LIN {X 0,Y 171.368,Z 489.651,A -85,B 0,C 180,E1 -22896.483,E2 -22896.483} C_VEL
LIN {X 0,Y 171.436,Z 490.117,A -85,B 0,C 180,E1 -22897.2,E2 -22897.2} C_VEL
LIN {X 0,Y 172.205,Z 492.194,A -85,B 0,C 180,E1 -22897.901,E2 -22897.901} C_VEL
LIN {X 0,Y 174.178,Z 494.48,A -85,B 0,C 180,E1 -22898.881,E2 -22898.881} C_VEL
LIN {X 0,Y 175.074,Z 495.303,A -85,B 0,C 180,E1 -22899.298,E2 -22899.298} C_VEL
LIN {X 0,Y 177.261,Z 498.704,A -85,B 0,C 180,E1 -22900.369,E2 -22900.369} C_VEL
LIN {X 0,Y 178.749,Z 500.495,A -85,B 0,C 180,E1 -22901.039,E2 -22901.039} C_VEL
LIN {X 0,Y 181.276,Z 503.935,A -85,B 0,C 180,E1 -22902.154,E2 -22902.154} C_VEL
LIN {X 0,Y 189.16,Z 515.818,A -85,B 0,C 180,E1 -22905.372,E2 -22905.372} C_VEL
LIN {X 0,Y 196.547,Z 528.551,A -85,B 0,C 180,E1 -22908.092,E2 -22908.092} C_VEL
LIN {X 0,Y 202.891,Z 541.51,A -85,B 0,C 180,E1 -22910.279,E2 -22910.279} C_VEL
LIN {X 0,Y 211.2,Z 559.373,A -85,B 0,C 180,E1 -22912.892,E2 -22912.892} C_VEL
LIN {X 0,Y 219.957,Z 574.029,A -85,B 0,C 180,E1 -22915.185,E2 -22915.185} C_VEL
LIN {X 0,Y 227.98,Z 585.278,A -85,B 0,C 180,E1 -22917.037,E2 -22917.037} C_VEL
LIN {X 0,Y 236.394,Z 595.667,A -85,B 0,C 180,E1 -22918.93,E2 -22918.93} C_VEL
LIN {X 0,Y 244.254,Z 604.497,A -85,B 0,C 180,E1 -22920.716,E2 -22920.716} C_VEL
LIN {X 0,Y 253.064,Z 613.517,A -85,B 0,C 180,E1 -22922.703,E2 -22922.703} C_VEL
LIN {X 0,Y 263.679,Z 622.944,A -85,B 0,C 180,E1 -22924.981,E2 -22924.981} C_VEL
LIN {X 0,Y 276.705,Z 633.025,A -85,B 0,C 180,E1 -22927.606,E2 -22927.606} C_VEL
LIN {X 0,Y 290.949,Z 643.204,A -85,B 0,C 180,E1 -22930.392,E2 -22930.392} C_VEL
LIN {X 0,Y 299.892,Z 649.736,A -85,B 0,C 180,E1 -22932.263,E2 -22932.263} C_VEL
LIN {X 0,Y 305.097,Z 653.329,A -85,B 0,C 180,E1 -22933.434,E2 -22933.434} C_VEL
LIN {X 0,Y 312.329,Z 658.424,A -85,B 0,C 180,E1 -22935.36,E2 -22935.36} C_VEL
LIN {X 0,Y 318.766,Z 662.437,A -85,B 0,C 180,E1 -22937.263,E2 -22937.263} C_VEL
LIN {X 0,Y 322.744,Z 665.158,A -85,B 0,C 180,E1 -22938.698,E2 -22938.698} C_VEL
LIN {X 0,Y 327.506,Z 668.458,A -85,B 0,C 180,E1 -22940.777,E2 -22940.777} C_VEL
LIN {X 0,Y 331.235,Z 670.635,A -85,B 0,C 180,E1 -22942.686,E2 -22942.686} C_VEL
LIN {X 0,Y 333.377,Z 671.715,A -85,B 0,C 180,E1 -22943.95,E2 -22943.95} C_VEL
LIN {X 0,Y 335.116,Z 672.498,A -85,B 0,C 180,E1 -22945.188,E2 -22945.188} C_VEL
LIN {X 0,Y 336.568,Z 673.013,A -85,B 0,C 180,E1 -22946.408,E2 -22946.408} C_VEL
LIN {X 0,Y 337.598,Z 673.448,A -85,B 0,C 180,E1 -22947.711,E2 -22947.711} C_VEL
LIN {X 0,Y 338.318,Z 673.7,A -85,B 0,C 180,E1 -22950,E2 -22950} C_VEL
LIN {X 0,Y 338.036,Z 673.676,A -85,B 0,C 180,E1 -22951.191,E2 -22951.191} C_VEL
LIN {X 0,Y 337.502,Z 673.41,A -85,B 0,C 180,E1 -22952.387,E2 -22952.387} C_VEL
LIN {X 0,Y 336.558,Z 672.994,A -85,B 0,C 180,E1 -22953.592,E2 -22953.592} C_VEL
LIN {X 0,Y 335.084,Z 672.488,A -85,B 0,C 180,E1 -22954.812,E2 -22954.812} C_VEL
LIN {X 0,Y 332.493,Z 671.329,A -85,B 0,C 180,E1 -22956.583,E2 -22956.583} C_VEL
LIN {X 0,Y 328.728,Z 669.23,A -85,B 0,C 180,E1 -22958.607,E2 -22958.607} C_VEL
LIN {X 0,Y 324.566,Z 666.489,A -85,B 0,C 180,E1 -22960.529,E2 -22960.529} C_VEL
LIN {X 0,Y 321.225,Z 664.079,A -85,B 0,C 180,E1 -22961.884,E2 -22961.884} C_VEL
LIN {X 0,Y 317.5,Z 661.727,A -85,B 0,C 180,E1 -22963.116,E2 -22963.116} C_VEL
LIN {X 0,Y 312.33,Z 658.43,A -85,B 0,C 180,E1 -22964.64,E2 -22964.64} C_VEL
LIN {X 0,Y 307.138,Z 654.773,A -85,B 0,C 180,E1 -22966.053,E2 -22966.053} C_VEL
LIN {X 0,Y 300.05,Z 649.811,A -85,B 0,C 180,E1 -22967.728,E2 -22967.728} C_VEL
LIN {X 0,Y 289.754,Z 642.358,A -85,B 0,C 180,E1 -22969.85,E2 -22969.85} C_VEL
LIN {X 0,Y 274.478,Z 631.398,A -85,B 0,C 180,E1 -22972.82,E2 -22972.82} C_VEL
LIN {X 0,Y 261.571,Z 621.184,A -85,B 0,C 180,E1 -22975.461,E2 -22975.461} C_VEL
LIN {X 0,Y 249.201,Z 609.815,A -85,B 0,C 180,E1 -22978.147,E2 -22978.147} C_VEL
LIN {X 0,Y 238.841,Z 598.535,A -85,B 0,C 180,E1 -22980.508,E2 -22980.508} C_VEL
LIN {X 0,Y 230.498,Z 588.456,A -85,B 0,C 180,E1 -22982.419,E2 -22982.419} C_VEL
LIN {X 0,Y 222.857,Z 578.314,A -85,B 0,C 180,E1 -22984.131,E2 -22984.131} C_VEL
LIN {X 0,Y 214.033,Z 564.466,A -85,B 0,C 180,E1 -22986.324,E2 -22986.324} C_VEL
LIN {X 0,Y 207.085,Z 551.017,A -85,B 0,C 180,E1 -22988.343,E2 -22988.343} C_VEL
LIN {X 0,Y 200.045,Z 535.481,A -85,B 0,C 180,E1 -22990.686,E2 -22990.686} C_VEL
LIN {X 0,Y 193.982,Z 523.965,A -85,B 0,C 180,E1 -22992.824,E2 -22992.824} C_VEL
LIN {X 0,Y 186.911,Z 512.312,A -85,B 0,C 180,E1 -22995.505,E2 -22995.505} C_VEL
LIN {X 0,Y 180.667,Z 503.29,A -85,B 0,C 180,E1 -22998.099,E2 -22998.099} C_VEL
LIN {X 0,Y 177.863,Z 499.314,A -85,B 0,C 180,E1 -22999.364,E2 -22999.364} C_VEL
LIN {X 0,Y 175.532,Z 496.228,A -85,B 0,C 180,E1 -23000.46,E2 -23000.46} C_VEL
LIN {X 0,Y 174.788,Z 494.891,A -85,B 0,C 180,E1 -23000.844,E2 -23000.844} C_VEL
LIN {X 0,Y 172.504,Z 492.69,A -85,B 0,C 180,E1 -23001.938,E2 -23001.938} C_VEL
LIN {X 0,Y 171.499,Z 490.425,A -85,B 0,C 180,E1 -23002.631,E2 -23002.631} C_VEL
LIN {X 0,Y 171.377,Z 489.669,A -85,B 0,C 180,E1 -23003.336,E2 -23003.336} C_VEL
LIN {X 0,Y 171.381,Z 489.625,A -85,B 0,C 180,E1 -23007.789,E2 -23007.789} C_VEL
LIN {X 0,Y 171.384,Z 489.611,A -85,B 0,C 180,E1 -23010.527,E2 -23010.527} C_VEL
LIN {X 0,Y 171.396,Z 489.63,A -85,B 0,C 180,E1 -23015.797,E2 -23015.797} C_VEL
LIN {X 0,Y 171.502,Z 489.574,A -85,B 0,C 180,E1 -23020.867,E2 -23020.867} C_VEL
LIN {X 0,Y 171.541,Z 489.614,A -85,B 0,C 180,E1 -23025.774,E2 -23025.774} C_VEL
LIN {X 0,Y 171.838,Z 489.529,A -85,B 0,C 180,E1 -23030.588,E2 -23030.588} C_VEL
LIN {X 0,Y 171.774,Z 489.585,A -85,B 0,C 180,E1 -23035.31,E2 -23035.31} C_VEL
LIN {X 0,Y 172.303,Z 489.467,A -85,B 0,C 180,E1 -23040.004,E2 -23040.004} C_VEL
LIN {X 0,Y 171.775,Z 489.588,A -85,B 0,C 180,E1 -23044.697,E2 -23044.697} C_VEL
LIN {X 0,Y 171.84,Z 489.524,A -85,B 0,C 180,E1 -23049.419,E2 -23049.419} C_VEL
LIN {X 0,Y 171.529,Z 489.615,A -85,B 0,C 180,E1 -23054.235,E2 -23054.235} C_VEL
LIN {X 0,Y 171.476,Z 489.578,A -85,B 0,C 180,E1 -23059.498,E2 -23059.498} C_VEL
LIN {X 0,Y 171.404,Z 489.596,A -85,B 0,C 180,E1 -23065.571,E2 -23065.571} C_VEL
LIN {X 0,Y 171.409,Z 489.635,A -85,B 0,C 180,E1 -23070.569,E2 -23070.569} C_VEL
LIN {X 0,Y 171.404,Z 489.723,A -85,B 0,C 180,E1 -23076.301,E2 -23076.301} C_VEL
LIN {X 0,Y 171.544,Z 490.53,A -85,B 0,C 180,E1 -23076.998,E2 -23076.998} C_VEL
LIN {X 0,Y 173.033,Z 493.38,A -85,B 0,C 180,E1 -23077.943,E2 -23077.943} C_VEL
LIN {X 0,Y 175.65,Z 496.732,A -85,B 0,C 180,E1 -23079.23,E2 -23079.23} C_VEL
LIN {X 0,Y 179.466,Z 502.8,A -85,B 0,C 180,E1 -23081.051,E2 -23081.051} C_VEL
LIN {X 0,Y 182.698,Z 508.235,A -85,B 0,C 180,E1 -23082.504,E2 -23082.504} C_VEL
LIN {X 0,Y 189.282,Z 520.227,A -85,B 0,C 180,E1 -23085.251,E2 -23085.251} C_VEL
LIN {X 0,Y 194.403,Z 531.098,A -85,B 0,C 180,E1 -23087.255,E2 -23087.255} C_VEL
LIN {X 0,Y 199.319,Z 543.1,A -85,B 0,C 180,E1 -23089.1,E2 -23089.1} C_VEL
LIN {X 0,Y 200.075,Z 545.841,A -85,B 0,C 180,E1 -23089.413,E2 -23089.413} C_VEL
LIN {X 0,Y 201.512,Z 556.425,A -85,B 0,C 180,E1 -23090.24,E2 -23090.24} C_VEL
LIN {X 0,Y 199.145,Z 597.614,A -85,B 0,C 180,E1 -23091.634,E2 -23091.634} C_VEL
LIN {X 0,Y 197.92,Z 608.393,A -85,B 0,C 180,E1 -23092.223,E2 -23092.223} C_VEL
LIN {X 0,Y 196.28,Z 618.373,A -85,B 0,C 180,E1 -23092.988,E2 -23092.988} C_VEL
LIN {X 0,Y 194.704,Z 626.202,A -85,B 0,C 180,E1 -23093.767,E2 -23093.767} C_VEL
LIN {X 0,Y 192.484,Z 635.344,A -85,B 0,C 180,E1 -23094.896,E2 -23094.896} C_VEL
LIN {X 0,Y 189.963,Z 644.341,A -85,B 0,C 180,E1 -23096.293,E2 -23096.293} C_VEL
LIN {X 0,Y 187.212,Z 653.065,A -85,B 0,C 180,E1 -23097.978,E2 -23097.978} C_VEL
LIN {X 0,Y 184.639,Z 660.483,A -85,B 0,C 180,E1 -23099.713,E2 -23099.713} C_VEL
LIN {X 0,Y 181.263,Z 669.275,A -85,B 0,C 180,E1 -23102.273,E2 -23102.273} C_VEL
LIN {X 0,Y 178.969,Z 675.267,A -85,B 0,C 180,E1 -23104.408,E2 -23104.408} C_VEL
LIN {X 0,Y 176.436,Z 681.58,A -85,B 0,C 180,E1 -23107.147,E2 -23107.147} C_VEL
LIN {X 0,Y 174.148,Z 686.853,A -85,B 0,C 180,E1 -23109.939,E2 -23109.939} C_VEL
LIN {X 0,Y 171.881,Z 691.945,A -85,B 0,C 180,E1 -23113.368,E2 -23113.368} C_VEL
LIN {X 0,Y 170.408,Z 695.916,A -85,B 0,C 180,E1 -23116.889,E2 -23116.889} C_VEL
LIN {X 0,Y 169.423,Z 698.857,A -85,B 0,C 180,E1 -23120.449,E2 -23120.449} C_VEL
LIN {X 0,Y 169.021,Z 700.362,A -85,B 0,C 180,E1 -23122.834,E2 -23122.834} C_VEL
LIN {X 0,Y 168.867,Z 701.898,A -85,B 0,C 180,E1 -23127.615,E2 -23127.615} C_VEL
LIN {X 0,Y 168.971,Z 702.182,A -85,B 0,C 180,E1 -23130,E2 -23130} C_VEL
LIN {X 0,Y 168.87,Z 701.296,A -85,B 0,C 180,E1 -23134.775,E2 -23134.775} C_VEL
LIN {X 0,Y 168.877,Z 701.169,A -85,B 0,C 180,E1 -23135.1,E2 -23135.1} C_VEL
LIN {X 0,Y 168.342,Z 700.396,A -85,B 0,C 180,E1 -23137.08,E2 -23137.08} C_VEL
LIN {X 0,Y 166.004,Z 698.459,A -85,B 0,C 180,E1 -23140.328,E2 -23140.328} C_VEL
LIN {X 0,Y 164.302,Z 696.463,A -85,B 0,C 180,E1 -23142.94,E2 -23142.94} C_VEL
LIN {X 0,Y 163.985,Z 694.593,A -85,B 0,C 180,E1 -23144.901,E2 -23144.901} C_VEL
LIN {X 0,Y 164.176,Z 693.859,A -85,B 0,C 180,E1 -23145.542,E2 -23145.542} C_VEL
LIN {X 0,Y 165.829,Z 690.235,A -85,B 0,C 180,E1 -23148.533,E2 -23148.533} C_VEL
LIN {X 0,Y 168.314,Z 684.658,A -85,B 0,C 180,E1 -23152.073,E2 -23152.073} C_VEL
LIN {X 0,Y 171.157,Z 678.377,A -85,B 0,C 180,E1 -23155.202,E2 -23155.202} C_VEL
LIN {X 0,Y 173.767,Z 672.201,A -85,B 0,C 180,E1 -23157.717,E2 -23157.717} C_VEL
LIN {X 0,Y 177.073,Z 663.985,A -85,B 0,C 180,E1 -23160.4,E2 -23160.4} C_VEL
LIN {X 0,Y 180.029,Z 656.162,A -85,B 0,C 180,E1 -23162.464,E2 -23162.464} C_VEL
LIN {X 0,Y 182.892,Z 648.084,A -85,B 0,C 180,E1 -23164.193,E2 -23164.193} C_VEL
LIN {X 0,Y 185.844,Z 638.326,A -85,B 0,C 180,E1 -23165.884,E2 -23165.884} C_VEL
LIN {X 0,Y 188.077,Z 629.94,A -85,B 0,C 180,E1 -23167.052,E2 -23167.052} C_VEL
LIN {X 0,Y 190.391,Z 619.437,A -85,B 0,C 180,E1 -23168.192,E2 -23168.192} C_VEL
LIN {X 0,Y 192.229,Z 609.145,A -85,B 0,C 180,E1 -23169.011,E2 -23169.011} C_VEL
LIN {X 0,Y 193.567,Z 598.773,A -85,B 0,C 180,E1 -23169.593,E2 -23169.593} C_VEL
LIN {X 0,Y 194.905,Z 576.946,A -85,B 0,C 180,E1 -23170.407,E2 -23170.407} C_VEL
LIN {X 0,Y 195.942,Z 556.279,A -85,B 0,C 180,E1 -23171.126,E2 -23171.126} C_VEL
LIN {X 0,Y 194.549,Z 547.053,A -85,B 0,C 180,E1 -23171.928,E2 -23171.928} C_VEL
LIN {X 0,Y 190.164,Z 535.964,A -85,B 0,C 180,E1 -23173.681,E2 -23173.681} C_VEL
LIN {X 0,Y 185.387,Z 525.465,A -85,B 0,C 180,E1 -23175.663,E2 -23175.663} C_VEL
LIN {X 0,Y 179.255,Z 513.895,A -85,B 0,C 180,E1 -23178.369,E2 -23178.369} C_VEL
LIN {X 0,Y 174.37,Z 505.581,A -85,B 0,C 180,E1 -23180.72,E2 -23180.72} C_VEL
LIN {X 0,Y 171.2,Z 500.576,A -85,B 0,C 180,E1 -23182.36,E2 -23182.36} C_VEL
LIN {X 0,Y 168.626,Z 497.072,A -85,B 0,C 180,E1 -23183.746,E2 -23183.746} C_VEL
LIN {X 0,Y 167.967,Z 495.868,A -85,B 0,C 180,E1 -23184.138,E2 -23184.138} C_VEL
LIN {X 0,Y 165.55,Z 493.655,A -85,B 0,C 180,E1 -23185.468,E2 -23185.468} C_VEL
LIN {X 0,Y 164.421,Z 491.155,A -85,B 0,C 180,E1 -23186.416,E2 -23186.416} C_VEL
LIN {X 0,Y 164.347,Z 490.531,A -85,B 0,C 180,E1 -23187.279,E2 -23187.279} C_VEL
LIN {X 0,Y 164.291,Z 490.484,A -85,B 0,C 180,E1 -23191.926,E2 -23191.926} C_VEL
LIN {X 0,Y 164.358,Z 490.475,A -85,B 0,C 180,E1 -23194.681,E2 -23194.681} C_VEL
LIN {X 0,Y 164.417,Z 490.459,A -85,B 0,C 180,E1 -23200.116,E2 -23200.116} C_VEL
LIN {X 0,Y 164.46,Z 490.486,A -85,B 0,C 180,E1 -23205.14,E2 -23205.14} C_VEL
LIN {X 0,Y 164.759,Z 490.406,A -85,B 0,C 180,E1 -23210.172,E2 -23210.172} C_VEL
LIN {X 0,Y 164.814,Z 490.411,A -85,B 0,C 180,E1 -23212.647,E2 -23212.647} C_VEL
LIN {X 0,Y 165.268,Z 490.343,A -85,B 0,C 180,E1 -23219.996,E2 -23219.996} C_VEL
LIN {X 0,Y 164.813,Z 490.425,A -85,B 0,C 180,E1 -23227.346,E2 -23227.346} C_VEL
LIN {X 0,Y 164.697,Z 490.418,A -85,B 0,C 180,E1 -23231.053,E2 -23231.053} C_VEL
LIN {X 0,Y 164.422,Z 490.466,A -85,B 0,C 180,E1 -23237.406,E2 -23237.406} C_VEL
LIN {X 0,Y 164.414,Z 490.458,A -85,B 0,C 180,E1 -23239.992,E2 -23239.992} C_VEL
LIN {X 0,Y 164.328,Z 490.482,A -85,B 0,C 180,E1 -23246.088,E2 -23246.088} C_VEL
LIN {X 0,Y 164.348,Z 490.498,A -85,B 0,C 180,E1 -23252.362,E2 -23252.362} C_VEL
LIN {X 0,Y 164.353,Z 490.85,A -85,B 0,C 180,E1 -23253.768,E2 -23253.768} C_VEL
LIN {X 0,Y 164.764,Z 492.175,A -85,B 0,C 180,E1 -23254.394,E2 -23254.394} C_VEL
LIN {X 0,Y 166.406,Z 494.696,A -85,B 0,C 180,E1 -23255.421,E2 -23255.421} C_VEL
LIN {X 0,Y 168.271,Z 496.336,A -85,B 0,C 180,E1 -23256.426,E2 -23256.426} C_VEL
LIN {X 0,Y 170.442,Z 499.713,A -85,B 0,C 180,E1 -23257.641,E2 -23257.641} C_VEL
LIN {X 0,Y 172.014,Z 501.392,A -85,B 0,C 180,E1 -23258.43,E2 -23258.43} C_VEL
LIN {X 0,Y 174.717,Z 505.136,A -85,B 0,C 180,E1 -23259.779,E2 -23259.779} C_VEL
LIN {X 0,Y 181.198,Z 514.584,A -85,B 0,C 180,E1 -23262.742,E2 -23262.742} C_VEL
LIN {X 0,Y 187.188,Z 524.201,A -85,B 0,C 180,E1 -23265.216,E2 -23265.216} C_VEL
LIN {X 0,Y 193.294,Z 535.317,A -85,B 0,C 180,E1 -23267.55,E2 -23267.55} C_VEL
LIN {X 0,Y 199.394,Z 548.354,A -85,B 0,C 180,E1 -23269.751,E2 -23269.751} C_VEL
LIN {X 0,Y 206.259,Z 563.313,A -85,B 0,C 180,E1 -23272.01,E2 -23272.01} C_VEL
LIN {X 0,Y 215.082,Z 578.411,A -85,B 0,C 180,E1 -23274.447,E2 -23274.447} C_VEL
LIN {X 0,Y 223.661,Z 590.654,A -85,B 0,C 180,E1 -23276.575,E2 -23276.575} C_VEL
LIN {X 0,Y 233.242,Z 602.662,A -85,B 0,C 180,E1 -23278.992,E2 -23278.992} C_VEL
LIN {X 0,Y 242.719,Z 613.234,A -85,B 0,C 180,E1 -23281.369,E2 -23281.369} C_VEL
LIN {X 0,Y 253.99,Z 624.019,A -85,B 0,C 180,E1 -23284.057,E2 -23284.057} C_VEL
LIN {X 0,Y 267.246,Z 634.657,A -85,B 0,C 180,E1 -23286.981,E2 -23286.981} C_VEL
LIN {X 0,Y 280.808,Z 644.286,A -85,B 0,C 180,E1 -23289.797,E2 -23289.797} C_VEL
LIN {X 0,Y 289.669,Z 650.424,A -85,B 0,C 180,E1 -23291.615,E2 -23291.615} C_VEL
LIN {X 0,Y 298.756,Z 656.783,A -85,B 0,C 180,E1 -23293.603,E2 -23293.603} C_VEL
LIN {X 0,Y 305.451,Z 661.513,A -85,B 0,C 180,E1 -23295.339,E2 -23295.339} C_VEL
LIN {X 0,Y 311.049,Z 665.144,A -85,B 0,C 180,E1 -23296.942,E2 -23296.942} C_VEL
LIN {X 0,Y 315.659,Z 668.041,A -85,B 0,C 180,E1 -23298.441,E2 -23298.441} C_VEL
LIN {X 0,Y 320.614,Z 671.559,A -85,B 0,C 180,E1 -23300.531,E2 -23300.531} C_VEL
LIN {X 0,Y 324.673,Z 674.038,A -85,B 0,C 180,E1 -23302.538,E2 -23302.538} C_VEL
LIN {X 0,Y 326.939,Z 675.216,A -85,B 0,C 180,E1 -23303.83,E2 -23303.83} C_VEL
LIN {X 0,Y 328.818,Z 676.119,A -85,B 0,C 180,E1 -23305.096,E2 -23305.096} C_VEL
LIN {X 0,Y 330.815,Z 676.869,A -85,B 0,C 180,E1 -23306.805,E2 -23306.805} C_VEL
LIN {X 0,Y 331.94,Z 677.388,A -85,B 0,C 180,E1 -23308.787,E2 -23308.787} C_VEL
LIN {X 0,Y 332.268,Z 677.395,A -85,B 0,C 180,E1 -23310,E2 -23310} C_VEL
LIN {X 0,Y 331.956,Z 677.37,A -85,B 0,C 180,E1 -23311.213,E2 -23311.213} C_VEL
LIN {X 0,Y 330.815,Z 676.878,A -85,B 0,C 180,E1 -23313.195,E2 -23313.195} C_VEL
LIN {X 0,Y 328.794,Z 676.11,A -85,B 0,C 180,E1 -23314.905,E2 -23314.905} C_VEL
LIN {X 0,Y 325.649,Z 674.584,A -85,B 0,C 180,E1 -23316.926,E2 -23316.926} C_VEL
LIN {X 0,Y 322.062,Z 672.504,A -85,B 0,C 180,E1 -23318.786,E2 -23318.786} C_VEL
LIN {X 0,Y 319.06,Z 670.533,A -85,B 0,C 180,E1 -23320.149,E2 -23320.149} C_VEL
LIN {X 0,Y 315.62,Z 668.068,A -85,B 0,C 180,E1 -23321.561,E2 -23321.561} C_VEL
LIN {X 0,Y 310.432,Z 664.788,A -85,B 0,C 180,E1 -23323.233,E2 -23323.233} C_VEL
LIN {X 0,Y 305.192,Z 661.373,A -85,B 0,C 180,E1 -23324.73,E2 -23324.73} C_VEL
LIN {X 0,Y 298.775,Z 656.763,A -85,B 0,C 180,E1 -23326.396,E2 -23326.396} C_VEL
LIN {X 0,Y 287.857,Z 649.115,A -85,B 0,C 180,E1 -23328.777,E2 -23328.777} C_VEL
LIN {X 0,Y 274.845,Z 640.119,A -85,B 0,C 180,E1 -23331.433,E2 -23331.433} C_VEL
LIN {X 0,Y 261.888,Z 630.524,A -85,B 0,C 180,E1 -23334.165,E2 -23334.165} C_VEL
LIN {X 0,Y 250.241,Z 620.543,A -85,B 0,C 180,E1 -23336.83,E2 -23336.83} C_VEL
LIN {X 0,Y 241.128,Z 611.5,A -85,B 0,C 180,E1 -23339.034,E2 -23339.034} C_VEL
LIN {X 0,Y 230.967,Z 599.971,A -85,B 0,C 180,E1 -23341.576,E2 -23341.576} C_VEL
LIN {X 0,Y 221.735,Z 588.081,A -85,B 0,C 180,E1 -23343.905,E2 -23343.905} C_VEL
LIN {X 0,Y 211.545,Z 572.787,A -85,B 0,C 180,E1 -23346.479,E2 -23346.479} C_VEL
LIN {X 0,Y 204.033,Z 558.817,A -85,B 0,C 180,E1 -23348.682,E2 -23348.682} C_VEL
LIN {X 0,Y 195.443,Z 539.676,A -85,B 0,C 180,E1 -23351.661,E2 -23351.661} C_VEL
LIN {X 0,Y 189.813,Z 528.782,A -85,B 0,C 180,E1 -23353.761,E2 -23353.761} C_VEL
LIN {X 0,Y 182.873,Z 517.082,A -85,B 0,C 180,E1 -23356.549,E2 -23356.549} C_VEL
LIN {X 0,Y 177.001,Z 508.481,A -85,B 0,C 180,E1 -23359.131,E2 -23359.131} C_VEL
LIN {X 0,Y 174.344,Z 504.736,A -85,B 0,C 180,E1 -23360.395,E2 -23360.395} C_VEL
LIN {X 0,Y 171.31,Z 500.527,A -85,B 0,C 180,E1 -23361.927,E2 -23361.927} C_VEL
LIN {X 0,Y 169.042,Z 497.785,A -85,B 0,C 180,E1 -23363.118,E2 -23363.118} C_VEL
LIN {X 0,Y 167.93,Z 495.858,A -85,B 0,C 180,E1 -23363.767,E2 -23363.767} C_VEL
LIN {X 0,Y 165.685,Z 493.84,A -85,B 0,C 180,E1 -23364.998,E2 -23364.998} C_VEL
LIN {X 0,Y 164.419,Z 491.07,A -85,B 0,C 180,E1 -23366.041,E2 -23366.041} C_VEL
LIN {X 0,Y 164.314,Z 490.518,A -85,B 0,C 180,E1 -23366.929,E2 -23366.929} C_VEL
LIN {X 0,Y 164.349,Z 490.51,A -85,B 0,C 180,E1 -23369.131,E2 -23369.131} C_VEL
LIN {X 0,Y 164.349,Z 490.487,A -85,B 0,C 180,E1 -23374.688,E2 -23374.688} C_VEL
LIN {X 0,Y 164.411,Z 490.458,A -85,B 0,C 180,E1 -23380.121,E2 -23380.121} C_VEL
LIN {X 0,Y 164.469,Z 490.499,A -85,B 0,C 180,E1 -23385.148,E2 -23385.148} C_VEL
LIN {X 0,Y 164.759,Z 490.408,A -85,B 0,C 180,E1 -23390.18,E2 -23390.18} C_VEL
LIN {X 0,Y 164.813,Z 490.425,A -85,B 0,C 180,E1 -23392.654,E2 -23392.654} C_VEL
LIN {X 0,Y 165.268,Z 490.343,A -85,B 0,C 180,E1 -23400.004,E2 -23400.004} C_VEL
LIN {X 0,Y 164.814,Z 490.411,A -85,B 0,C 180,E1 -23407.353,E2 -23407.353} C_VEL
LIN {X 0,Y 164.696,Z 490.423,A -85,B 0,C 180,E1 -23411.051,E2 -23411.051} C_VEL
LIN {X 0,Y 164.417,Z 490.455,A -85,B 0,C 180,E1 -23417.414,E2 -23417.414} C_VEL
LIN {X 0,Y 164.42,Z 490.46,A -85,B 0,C 180,E1 -23420,E2 -23420} C_VEL
LIN {X 0,Y 164.338,Z 490.473,A -85,B 0,C 180,E1 -23426.095,E2 -23426.095} C_VEL
LIN {X 0,Y 164.36,Z 490.509,A -85,B 0,C 180,E1 -23432.369,E2 -23432.369} C_VEL
LIN {X 0,Y 164.371,Z 490.912,A -85,B 0,C 180,E1 -23433.419,E2 -23433.419} C_VEL
LIN {X 0,Y 164.852,Z 492.387,A -85,B 0,C 180,E1 -23434.075,E2 -23434.075} C_VEL
LIN {X 0,Y 166.509,Z 494.761,A -85,B 0,C 180,E1 -23435.087,E2 -23435.087} C_VEL
LIN {X 0,Y 168.197,Z 496.151,A -85,B 0,C 180,E1 -23435.99,E2 -23435.99} C_VEL
LIN {X 0,Y 170.237,Z 499.459,A -85,B 0,C 180,E1 -23437.145,E2 -23437.145} C_VEL
LIN {X 0,Y 172.277,Z 502.221,A -85,B 0,C 180,E1 -23438.207,E2 -23438.207} C_VEL
LIN {X 0,Y 176.131,Z 508.451,A -85,B 0,C 180,E1 -23440.148,E2 -23440.148} C_VEL
LIN {X 0,Y 180.462,Z 516.016,A -85,B 0,C 180,E1 -23442.181,E2 -23442.181} C_VEL
LIN {X 0,Y 186.936,Z 528.657,A -85,B 0,C 180,E1 -23444.987,E2 -23444.987} C_VEL
LIN {X 0,Y 192.82,Z 542.334,A -85,B 0,C 180,E1 -23447.379,E2 -23447.379} C_VEL
LIN {X 0,Y 194.799,Z 548.007,A -85,B 0,C 180,E1 -23448.184,E2 -23448.184} C_VEL
LIN {X 0,Y 196.004,Z 556.741,A -85,B 0,C 180,E1 -23448.912,E2 -23448.912} C_VEL
LIN {X 0,Y 193.657,Z 597.26,A -85,B 0,C 180,E1 -23450.326,E2 -23450.326} C_VEL
LIN {X 0,Y 192.397,Z 608.063,A -85,B 0,C 180,E1 -23450.923,E2 -23450.923} C_VEL
LIN {X 0,Y 190.875,Z 616.913,A -85,B 0,C 180,E1 -23451.587,E2 -23451.587} C_VEL
LIN {X 0,Y 189.006,Z 626.005,A -85,B 0,C 180,E1 -23452.491,E2 -23452.491} C_VEL
LIN {X 0,Y 186.706,Z 635.147,A -85,B 0,C 180,E1 -23453.64,E2 -23453.64} C_VEL
LIN {X 0,Y 184.091,Z 644.145,A -85,B 0,C 180,E1 -23455.065,E2 -23455.065} C_VEL
LIN {X 0,Y 181.225,Z 652.868,A -85,B 0,C 180,E1 -23456.786,E2 -23456.786} C_VEL
LIN {X 0,Y 178.516,Z 660.286,A -85,B 0,C 180,E1 -23458.558,E2 -23458.558} C_VEL
LIN {X 0,Y 174.988,Z 669.078,A -85,B 0,C 180,E1 -23461.187,E2 -23461.187} C_VEL
LIN {X 0,Y 172.568,Z 675.07,A -85,B 0,C 180,E1 -23463.386,E2 -23463.386} C_VEL
LIN {X 0,Y 169.899,Z 681.384,A -85,B 0,C 180,E1 -23466.215,E2 -23466.215} C_VEL
LIN {X 0,Y 167.456,Z 686.656,A -85,B 0,C 180,E1 -23469.1,E2 -23469.1} C_VEL
LIN {X 0,Y 165.073,Z 691.749,A -85,B 0,C 180,E1 -23472.661,E2 -23472.661} C_VEL
LIN {X 0,Y 163.458,Z 695.719,A -85,B 0,C 180,E1 -23476.321,E2 -23476.321} C_VEL
LIN {X 0,Y 162.405,Z 698.66,A -85,B 0,C 180,E1 -23480.032,E2 -23480.032} C_VEL
LIN {X 0,Y 161.962,Z 700.165,A -85,B 0,C 180,E1 -23482.52,E2 -23482.52} C_VEL
LIN {X 0,Y 161.768,Z 701.701,A -85,B 0,C 180,E1 -23487.51,E2 -23487.51} C_VEL
LIN {X 0,Y 161.869,Z 701.985,A -85,B 0,C 180,E1 -23490,E2 -23490} C_VEL
LIN {X 0,Y 161.776,Z 701.099,A -85,B 0,C 180,E1 -23494.984,E2 -23494.984} C_VEL
LIN {X 0,Y 161.98,Z 700.166,A -85,B 0,C 180,E1 -23497.479,E2 -23497.479} C_VEL
LIN {X 0,Y 163.059,Z 696.81,A -85,B 0,C 180,E1 -23502.445,E2 -23502.445} C_VEL
LIN {X 0,Y 164.176,Z 693.859,A -85,B 0,C 180,E1 -23505.542,E2 -23505.542} C_VEL
LIN {X 0,Y 164.476,Z 691.704,A -85,B 0,C 180,E1 -23507.452,E2 -23507.452} C_VEL
LIN {X 0,Y 163.645,Z 687.755,A -85,B 0,C 180,E1 -23510.626,E2 -23510.626} C_VEL
LIN {X 0,Y 163.153,Z 683.225,A -85,B 0,C 180,E1 -23513.713,E2 -23513.713} C_VEL
LIN {X 0,Y 163.948,Z 680,A -85,B 0,C 180,E1 -23515.425,E2 -23515.425} C_VEL
LIN {X 0,Y 167.466,Z 672.003,A -85,B 0,C 180,E1 -23518.856,E2 -23518.856} C_VEL
LIN {X 0,Y 170.965,Z 663.789,A -85,B 0,C 180,E1 -23521.609,E2 -23521.609} C_VEL
LIN {X 0,Y 174.064,Z 655.965,A -85,B 0,C 180,E1 -23523.722,E2 -23523.722} C_VEL
LIN {X 0,Y 177.067,Z 647.888,A -85,B 0,C 180,E1 -23525.484,E2 -23525.484} C_VEL
LIN {X 0,Y 180.143,Z 638.13,A -85,B 0,C 180,E1 -23527.207,E2 -23527.207} C_VEL
LIN {X 0,Y 182.455,Z 629.743,A -85,B 0,C 180,E1 -23528.397,E2 -23528.397} C_VEL
LIN {X 0,Y 184.857,Z 619.241,A -85,B 0,C 180,E1 -23529.554,E2 -23529.554} C_VEL
LIN {X 0,Y 186.808,Z 608.823,A -85,B 0,C 180,E1 -23530.385,E2 -23530.385} C_VEL
LIN {X 0,Y 188.149,Z 598.632,A -85,B 0,C 180,E1 -23530.967,E2 -23530.967} C_VEL
LIN {X 0,Y 189.546,Z 576.839,A -85,B 0,C 180,E1 -23531.796,E2 -23531.796} C_VEL
LIN {X 0,Y 190.585,Z 557.523,A -85,B 0,C 180,E1 -23532.476,E2 -23532.476} C_VEL
LIN {X 0,Y 189.405,Z 549.639,A -85,B 0,C 180,E1 -23533.2,E2 -23533.2} C_VEL
LIN {X 0,Y 184.565,Z 537.416,A -85,B 0,C 180,E1 -23535.274,E2 -23535.274} C_VEL
LIN {X 0,Y 180.217,Z 527.991,A -85,B 0,C 180,E1 -23537.215,E2 -23537.215} C_VEL
LIN {X 0,Y 173.933,Z 515.984,A -85,B 0,C 180,E1 -23540.235,E2 -23540.235} C_VEL
LIN {X 0,Y 170.407,Z 510.142,A -85,B 0,C 180,E1 -23542.061,E2 -23542.061} C_VEL
LIN {X 0,Y 167.874,Z 506.005,A -85,B 0,C 180,E1 -23543.465,E2 -23543.465} C_VEL
LIN {X 0,Y 164.74,Z 501.67,A -85,B 0,C 180,E1 -23545.274,E2 -23545.274} C_VEL
LIN {X 0,Y 162.18,Z 498.652,A -85,B 0,C 180,E1 -23546.828,E2 -23546.828} C_VEL
LIN {X 0,Y 161.169,Z 496.857,A -85,B 0,C 180,E1 -23547.523,E2 -23547.523} C_VEL
LIN {X 0,Y 158.82,Z 494.949,A -85,B 0,C 180,E1 -23549.032,E2 -23549.032} C_VEL
LIN {X 0,Y 157.364,Z 492.026,A -85,B 0,C 180,E1 -23550.388,E2 -23550.388} C_VEL
LIN {X 0,Y 157.237,Z 491.432,A -85,B 0,C 180,E1 -23551.279,E2 -23551.279} C_VEL
LIN {X 0,Y 157.267,Z 491.377,A -85,B 0,C 180,E1 -23556.281,E2 -23556.281} C_VEL
LIN {X 0,Y 157.36,Z 491.341,A -85,B 0,C 180,E1 -23559.7,E2 -23559.7} C_VEL
LIN {X 0,Y 157.396,Z 491.35,A -85,B 0,C 180,E1 -23564.456,E2 -23564.456} C_VEL
LIN {X 0,Y 157.681,Z 491.289,A -85,B 0,C 180,E1 -23569.726,E2 -23569.726} C_VEL
LIN {X 0,Y 157.753,Z 491.285,A -85,B 0,C 180,E1 -23572.315,E2 -23572.315} C_VEL
LIN {X 0,Y 158.23,Z 491.218,A -85,B 0,C 180,E1 -23579.996,E2 -23579.996} C_VEL
LIN {X 0,Y 157.752,Z 491.298,A -85,B 0,C 180,E1 -23587.677,E2 -23587.677} C_VEL
LIN {X 0,Y 157.626,Z 491.299,A -85,B 0,C 180,E1 -23591.219,E2 -23591.219} C_VEL
LIN {X 0,Y 157.402,Z 491.371,A -85,B 0,C 180,E1 -23595.535,E2 -23595.535} C_VEL
LIN {X 0,Y 157.297,Z 491.351,A -85,B 0,C 180,E1 -23600.938,E2 -23600.938} C_VEL
LIN {X 0,Y 157.259,Z 491.358,A -85,B 0,C 180,E1 -23606.645,E2 -23606.645} C_VEL
LIN {X 0,Y 157.278,Z 491.657,A -85,B 0,C 180,E1 -23609.621,E2 -23609.621} C_VEL
LIN {X 0,Y 157.592,Z 492.786,A -85,B 0,C 180,E1 -23610.385,E2 -23610.385} C_VEL
LIN {X 0,Y 159.197,Z 495.38,A -85,B 0,C 180,E1 -23611.617,E2 -23611.617} C_VEL
LIN {X 0,Y 161.459,Z 497.163,A -85,B 0,C 180,E1 -23613.051,E2 -23613.051} C_VEL
LIN {X 0,Y 163.482,Z 500.487,A -85,B 0,C 180,E1 -23614.388,E2 -23614.388} C_VEL
LIN {X 0,Y 165.501,Z 502.633,A -85,B 0,C 180,E1 -23615.561,E2 -23615.561} C_VEL
LIN {X 0,Y 168.085,Z 506.198,A -85,B 0,C 180,E1 -23617.034,E2 -23617.034} C_VEL
LIN {X 0,Y 172.906,Z 512.986,A -85,B 0,C 180,E1 -23619.554,E2 -23619.554} C_VEL
LIN {X 0,Y 177.99,Z 520.544,A -85,B 0,C 180,E1 -23621.959,E2 -23621.959} C_VEL
LIN {X 0,Y 183.619,Z 529.846,A -85,B 0,C 180,E1 -23624.404,E2 -23624.404} C_VEL
LIN {X 0,Y 189.395,Z 540.762,A -85,B 0,C 180,E1 -23626.733,E2 -23626.733} C_VEL
LIN {X 0,Y 194.728,Z 552.601,A -85,B 0,C 180,E1 -23628.775,E2 -23628.775} C_VEL
LIN {X 0,Y 201.859,Z 568.247,A -85,B 0,C 180,E1 -23631.242,E2 -23631.242} C_VEL
LIN {X 0,Y 210.51,Z 583.179,A -85,B 0,C 180,E1 -23633.746,E2 -23633.746} C_VEL
LIN {X 0,Y 218.276,Z 594.692,A -85,B 0,C 180,E1 -23635.897,E2 -23635.897} C_VEL
LIN {X 0,Y 226.162,Z 605.048,A -85,B 0,C 180,E1 -23638.111,E2 -23638.111} C_VEL
LIN {X 0,Y 234.418,Z 614.641,A -85,B 0,C 180,E1 -23640.387,E2 -23640.387} C_VEL
LIN {X 0,Y 242.814,Z 623.364,A -85,B 0,C 180,E1 -23642.63,E2 -23642.63} C_VEL
LIN {X 0,Y 254.728,Z 633.732,A -85,B 0,C 180,E1 -23645.564,E2 -23645.564} C_VEL
LIN {X 0,Y 269.029,Z 644.182,A -85,B 0,C 180,E1 -23648.781,E2 -23648.781} C_VEL
LIN {X 0,Y 281.628,Z 652.561,A -85,B 0,C 180,E1 -23651.484,E2 -23651.484} C_VEL
LIN {X 0,Y 292.553,Z 660.061,A -85,B 0,C 180,E1 -23653.919,E2 -23653.919} C_VEL
LIN {X 0,Y 299.534,Z 664.986,A -85,B 0,C 180,E1 -23655.704,E2 -23655.704} C_VEL
LIN {X 0,Y 304.733,Z 668.357,A -85,B 0,C 180,E1 -23657.162,E2 -23657.162} C_VEL
LIN {X 0,Y 309.727,Z 671.52,A -85,B 0,C 180,E1 -23658.772,E2 -23658.772} C_VEL
LIN {X 0,Y 313.619,Z 674.292,A -85,B 0,C 180,E1 -23660.389,E2 -23660.389} C_VEL
LIN {X 0,Y 318.723,Z 677.455,A -85,B 0,C 180,E1 -23662.851,E2 -23662.851} C_VEL
LIN {X 0,Y 322.189,Z 679.196,A -85,B 0,C 180,E1 -23664.994,E2 -23664.994} C_VEL
LIN {X 0,Y 323.932,Z 679.922,A -85,B 0,C 180,E1 -23666.344,E2 -23666.344} C_VEL
LIN {X 0,Y 325.013,Z 680.344,A -85,B 0,C 180,E1 -23667.521,E2 -23667.521} C_VEL
LIN {X 0,Y 325.623,Z 680.637,A -85,B 0,C 180,E1 -23668.763,E2 -23668.763} C_VEL
LIN {X 0,Y 325.956,Z 680.664,A -85,B 0,C 180,E1 -23670,E2 -23670} C_VEL
LIN {X 0,Y 325.634,Z 680.624,A -85,B 0,C 180,E1 -23671.237,E2 -23671.237} C_VEL
LIN {X 0,Y 325.013,Z 680.333,A -85,B 0,C 180,E1 -23672.479,E2 -23672.479} C_VEL
LIN {X 0,Y 323.839,Z 679.87,A -85,B 0,C 180,E1 -23673.733,E2 -23673.733} C_VEL
LIN {X 0,Y 322.172,Z 679.197,A -85,B 0,C 180,E1 -23675.006,E2 -23675.006} C_VEL
LIN {X 0,Y 318.703,Z 677.482,A -85,B 0,C 180,E1 -23677.121,E2 -23677.121} C_VEL
LIN {X 0,Y 314.988,Z 675.237,A -85,B 0,C 180,E1 -23678.985,E2 -23678.985} C_VEL
LIN {X 0,Y 311.78,Z 673.038,A -85,B 0,C 180,E1 -23680.389,E2 -23680.389} C_VEL
LIN {X 0,Y 307.878,Z 670.331,A -85,B 0,C 180,E1 -23681.855,E2 -23681.855} C_VEL
LIN {X 0,Y 302.651,Z 667.041,A -85,B 0,C 180,E1 -23683.427,E2 -23683.427} C_VEL
LIN {X 0,Y 296.488,Z 662.798,A -85,B 0,C 180,E1 -23685.114,E2 -23685.114} C_VEL
LIN {X 0,Y 289.821,Z 658.167,A -85,B 0,C 180,E1 -23686.706,E2 -23686.706} C_VEL
LIN {X 0,Y 278.836,Z 650.743,A -85,B 0,C 180,E1 -23689.127,E2 -23689.127} C_VEL
LIN {X 0,Y 263.564,Z 640.349,A -85,B 0,C 180,E1 -23692.419,E2 -23692.419} C_VEL
LIN {X 0,Y 252.116,Z 631.599,A -85,B 0,C 180,E1 -23695.051,E2 -23695.051} C_VEL
LIN {X 0,Y 241.185,Z 621.822,A -85,B 0,C 180,E1 -23697.79,E2 -23697.79} C_VEL
LIN {X 0,Y 230.712,Z 610.495,A -85,B 0,C 180,E1 -23700.621,E2 -23700.621} C_VEL
LIN {X 0,Y 221.954,Z 599.646,A -85,B 0,C 180,E1 -23703.065,E2 -23703.065} C_VEL
LIN {X 0,Y 214.414,Z 589.166,A -85,B 0,C 180,E1 -23705.181,E2 -23705.181} C_VEL
LIN {X 0,Y 205.872,Z 575.535,A -85,B 0,C 180,E1 -23707.545,E2 -23707.545} C_VEL
LIN {X 0,Y 198.966,Z 562.296,A -85,B 0,C 180,E1 -23709.708,E2 -23709.708} C_VEL
LIN {X 0,Y 190.822,Z 543.776,A -85,B 0,C 180,E1 -23712.71,E2 -23712.71} C_VEL
LIN {X 0,Y 185.41,Z 533.084,A -85,B 0,C 180,E1 -23714.856,E2 -23714.856} C_VEL
LIN {X 0,Y 179.132,Z 522.27,A -85,B 0,C 180,E1 -23717.533,E2 -23717.533} C_VEL
LIN {X 0,Y 173.232,Z 513.452,A -85,B 0,C 180,E1 -23720.285,E2 -23720.285} C_VEL
LIN {X 0,Y 170.673,Z 509.812,A -85,B 0,C 180,E1 -23721.58,E2 -23721.58} C_VEL
LIN {X 0,Y 167.965,Z 506.081,A -85,B 0,C 180,E1 -23723.029,E2 -23723.029} C_VEL
LIN {X 0,Y 165.409,Z 502.425,A -85,B 0,C 180,E1 -23724.498,E2 -23724.498} C_VEL
LIN {X 0,Y 162.256,Z 498.764,A -85,B 0,C 180,E1 -23726.39,E2 -23726.39} C_VEL
LIN {X 0,Y 161.135,Z 496.856,A -85,B 0,C 180,E1 -23727.153,E2 -23727.153} C_VEL
LIN {X 0,Y 158.693,Z 494.791,A -85,B 0,C 180,E1 -23728.732,E2 -23728.732} C_VEL
LIN {X 0,Y 157.355,Z 491.978,A -85,B 0,C 180,E1 -23730.027,E2 -23730.027} C_VEL
LIN {X 0,Y 157.227,Z 491.408,A -85,B 0,C 180,E1 -23731.286,E2 -23731.286} C_VEL
LIN {X 0,Y 157.259,Z 491.397,A -85,B 0,C 180,E1 -23736.288,E2 -23736.288} C_VEL
LIN {X 0,Y 157.353,Z 491.338,A -85,B 0,C 180,E1 -23739.707,E2 -23739.707} C_VEL
LIN {X 0,Y 157.402,Z 491.371,A -85,B 0,C 180,E1 -23744.465,E2 -23744.465} C_VEL
LIN {X 0,Y 157.682,Z 491.288,A -85,B 0,C 180,E1 -23749.734,E2 -23749.734} C_VEL
LIN {X 0,Y 157.752,Z 491.298,A -85,B 0,C 180,E1 -23752.323,E2 -23752.323} C_VEL
LIN {X 0,Y 158.23,Z 491.218,A -85,B 0,C 180,E1 -23760.004,E2 -23760.004} C_VEL
LIN {X 0,Y 157.753,Z 491.285,A -85,B 0,C 180,E1 -23767.685,E2 -23767.685} C_VEL
LIN {X 0,Y 157.626,Z 491.304,A -85,B 0,C 180,E1 -23771.219,E2 -23771.219} C_VEL
LIN {X 0,Y 157.396,Z 491.35,A -85,B 0,C 180,E1 -23775.544,E2 -23775.544} C_VEL
LIN {X 0,Y 157.303,Z 491.357,A -85,B 0,C 180,E1 -23780.946,E2 -23780.946} C_VEL
LIN {X 0,Y 157.269,Z 491.352,A -85,B 0,C 180,E1 -23786.652,E2 -23786.652} C_VEL
LIN {X 0,Y 157.283,Z 491.658,A -85,B 0,C 180,E1 -23789.261,E2 -23789.261} C_VEL
LIN {X 0,Y 157.615,Z 492.844,A -85,B 0,C 180,E1 -23790.02,E2 -23790.02} C_VEL
LIN {X 0,Y 159.232,Z 495.422,A -85,B 0,C 180,E1 -23791.253,E2 -23791.253} C_VEL
LIN {X 0,Y 161.583,Z 497.458,A -85,B 0,C 180,E1 -23792.753,E2 -23792.753} C_VEL
LIN {X 0,Y 163.589,Z 500.569,A -85,B 0,C 180,E1 -23794.06,E2 -23794.06} C_VEL
LIN {X 0,Y 165.378,Z 502.391,A -85,B 0,C 180,E1 -23795.095,E2 -23795.095} C_VEL
LIN {X 0,Y 168.077,Z 506.278,A -85,B 0,C 180,E1 -23796.647,E2 -23796.647} C_VEL
LIN {X 0,Y 172.43,Z 513.44,A -85,B 0,C 180,E1 -23799.001,E2 -23799.001} C_VEL
LIN {X 0,Y 176.489,Z 520.707,A -85,B 0,C 180,E1 -23801.032,E2 -23801.032} C_VEL
LIN {X 0,Y 182.602,Z 532.892,A -85,B 0,C 180,E1 -23803.855,E2 -23803.855} C_VEL
LIN {X 0,Y 188.2,Z 546.423,A -85,B 0,C 180,E1 -23806.291,E2 -23806.291} C_VEL
LIN {X 0,Y 189.722,Z 550.794,A -85,B 0,C 180,E1 -23806.947,E2 -23806.947} C_VEL
LIN {X 0,Y 190.632,Z 558.719,A -85,B 0,C 180,E1 -23807.597,E2 -23807.597} C_VEL
LIN {X 0,Y 188.251,Z 597.07,A -85,B 0,C 180,E1 -23808.947,E2 -23808.947} C_VEL
LIN {X 0,Y 186.956,Z 607.807,A -85,B 0,C 180,E1 -23809.55,E2 -23809.55} C_VEL
LIN {X 0,Y 185.374,Z 616.718,A -85,B 0,C 180,E1 -23810.225,E2 -23810.225} C_VEL
LIN {X 0,Y 183.42,Z 625.809,A -85,B 0,C 180,E1 -23811.14,E2 -23811.14} C_VEL
LIN {X 0,Y 181.042,Z 634.951,A -85,B 0,C 180,E1 -23812.309,E2 -23812.309} C_VEL
LIN {X 0,Y 178.308,Z 643.948,A -85,B 0,C 180,E1 -23813.757,E2 -23813.757} C_VEL
LIN {X 0,Y 175.315,Z 652.672,A -85,B 0,C 180,E1 -23815.512,E2 -23815.512} C_VEL
LIN {X 0,Y 172.469,Z 660.089,A -85,B 0,C 180,E1 -23817.322,E2 -23817.322} C_VEL
LIN {X 0,Y 168.775,Z 668.881,A -85,B 0,C 180,E1 -23820.021,E2 -23820.021} C_VEL
LIN {X 0,Y 166.221,Z 674.873,A -85,B 0,C 180,E1 -23822.284,E2 -23822.284} C_VEL
LIN {X 0,Y 163.388,Z 681.186,A -85,B 0,C 180,E1 -23825.204,E2 -23825.204} C_VEL
LIN {X 0,Y 160.794,Z 686.458,A -85,B 0,C 180,E1 -23828.191,E2 -23828.191} C_VEL
LIN {X 0,Y 158.298,Z 691.552,A -85,B 0,C 180,E1 -23831.894,E2 -23831.894} C_VEL
LIN {X 0,Y 156.532,Z 695.522,A -85,B 0,C 180,E1 -23835.704,E2 -23835.704} C_VEL
LIN {X 0,Y 155.407,Z 698.464,A -85,B 0,C 180,E1 -23839.578,E2 -23839.578} C_VEL
LIN {X 0,Y 154.923,Z 699.969,A -85,B 0,C 180,E1 -23842.178,E2 -23842.178} C_VEL
LIN {X 0,Y 154.673,Z 701.505,A -85,B 0,C 180,E1 -23847.396,E2 -23847.396} C_VEL
LIN {X 0,Y 154.782,Z 701.789,A -85,B 0,C 180,E1 -23850,E2 -23850} C_VEL
LIN {X 0,Y 154.703,Z 700.903,A -85,B 0,C 180,E1 -23855.213,E2 -23855.213} C_VEL
LIN {X 0,Y 154.937,Z 699.969,A -85,B 0,C 180,E1 -23857.821,E2 -23857.821} C_VEL
LIN {X 0,Y 156.088,Z 696.613,A -85,B 0,C 180,E1 -23863.01,E2 -23863.01} C_VEL
LIN {X 0,Y 157.615,Z 692.981,A -85,B 0,C 180,E1 -23866.848,E2 -23866.848} C_VEL
LIN {X 0,Y 159.934,Z 688.249,A -85,B 0,C 180,E1 -23870.582,E2 -23870.582} C_VEL
LIN {X 0,Y 162.849,Z 682.279,A -85,B 0,C 180,E1 -23874.204,E2 -23874.204} C_VEL
LIN {X 0,Y 163.948,Z 680,A -85,B 0,C 180,E1 -23875.425,E2 -23875.425} C_VEL
LIN {X 0,Y 164.807,Z 676.605,A -85,B 0,C 180,E1 -23877.067,E2 -23877.067} C_VEL
LIN {X 0,Y 164.848,Z 670.82,A -85,B 0,C 180,E1 -23879.847,E2 -23879.847} C_VEL
LIN {X 0,Y 165.145,Z 664.579,A -85,B 0,C 180,E1 -23882.499,E2 -23882.499} C_VEL
LIN {X 0,Y 166.371,Z 660.272,A -85,B 0,C 180,E1 -23883.886,E2 -23883.886} C_VEL
LIN {X 0,Y 170.868,Z 649.003,A -85,B 0,C 180,E1 -23886.612,E2 -23886.612} C_VEL
LIN {X 0,Y 174.072,Z 639.523,A -85,B 0,C 180,E1 -23888.37,E2 -23888.37} C_VEL
LIN {X 0,Y 176.939,Z 629.547,A -85,B 0,C 180,E1 -23889.827,E2 -23889.827} C_VEL
LIN {X 0,Y 179.431,Z 619.044,A -85,B 0,C 180,E1 -23891,E2 -23891} C_VEL
LIN {X 0,Y 181.393,Z 609.039,A -85,B 0,C 180,E1 -23891.811,E2 -23891.811} C_VEL
LIN {X 0,Y 182.858,Z 597.896,A -85,B 0,C 180,E1 -23892.461,E2 -23892.461} C_VEL
LIN {X 0,Y 184.528,Z 573.459,A -85,B 0,C 180,E1 -23893.371,E2 -23893.371} C_VEL
LIN {X 0,Y 185.351,Z 558.629,A -85,B 0,C 180,E1 -23893.906,E2 -23893.906} C_VEL
LIN {X 0,Y 184.399,Z 552.465,A -85,B 0,C 180,E1 -23894.518,E2 -23894.518} C_VEL
LIN {X 0,Y 179.211,Z 539.178,A -85,B 0,C 180,E1 -23896.916,E2 -23896.916} C_VEL
LIN {X 0,Y 174.112,Z 528.451,A -85,B 0,C 180,E1 -23899.388,E2 -23899.388} C_VEL
LIN {X 0,Y 169.562,Z 519.798,A -85,B 0,C 180,E1 -23901.776,E2 -23901.776} C_VEL
LIN {X 0,Y 165.111,Z 512.074,A -85,B 0,C 180,E1 -23904.326,E2 -23904.326} C_VEL
LIN {X 0,Y 161.762,Z 507.476,A -85,B 0,C 180,E1 -23906.358,E2 -23906.358} C_VEL
LIN {X 0,Y 159.134,Z 504,A -85,B 0,C 180,E1 -23908.085,E2 -23908.085} C_VEL
LIN {X 0,Y 158.275,Z 502.9,A -85,B 0,C 180,E1 -23908.677,E2 -23908.677} C_VEL
LIN {X 0,Y 155.8,Z 500.269,A -85,B 0,C 180,E1 -23910.433,E2 -23910.433} C_VEL
LIN {X 0,Y 154.545,Z 497.966,A -85,B 0,C 180,E1 -23911.474,E2 -23911.474} C_VEL
LIN {X 0,Y 151.987,Z 496.1,A -85,B 0,C 180,E1 -23913.478,E2 -23913.478} C_VEL
LIN {X 0,Y 150.538,Z 493.71,A -85,B 0,C 180,E1 -23914.893,E2 -23914.893} C_VEL
LIN {X 0,Y 150.239,Z 492.531,A -85,B 0,C 180,E1 -23915.834,E2 -23915.834} C_VEL
LIN {X 0,Y 150.296,Z 492.211,A -85,B 0,C 180,E1 -23920.889,E2 -23920.889} C_VEL
LIN {X 0,Y 150.395,Z 492.243,A -85,B 0,C 180,E1 -23926.484,E2 -23926.484} C_VEL
LIN {X 0,Y 150.601,Z 492.173,A -85,B 0,C 180,E1 -23929.238,E2 -23929.238} C_VEL
LIN {X 0,Y 150.676,Z 492.163,A -85,B 0,C 180,E1 -23931.952,E2 -23931.952} C_VEL
LIN {X 0,Y 151.191,Z 492.094,A -85,B 0,C 180,E1 -23939.996,E2 -23939.996} C_VEL
LIN {X 0,Y 150.675,Z 492.173,A -85,B 0,C 180,E1 -23948.04,E2 -23948.04} C_VEL
LIN {X 0,Y 150.569,Z 492.178,A -85,B 0,C 180,E1 -23951.423,E2 -23951.423} C_VEL
LIN {X 0,Y 150.306,Z 492.238,A -85,B 0,C 180,E1 -23956.288,E2 -23956.288} C_VEL
LIN {X 0,Y 150.276,Z 492.222,A -85,B 0,C 180,E1 -23960.718,E2 -23960.718} C_VEL
LIN {X 0,Y 150.221,Z 492.544,A -85,B 0,C 180,E1 -23964.62,E2 -23964.62} C_VEL
LIN {X 0,Y 150.53,Z 493.696,A -85,B 0,C 180,E1 -23965.488,E2 -23965.488} C_VEL
LIN {X 0,Y 152.154,Z 496.309,A -85,B 0,C 180,E1 -23967.057,E2 -23967.057} C_VEL
LIN {X 0,Y 154.791,Z 498.354,A -85,B 0,C 180,E1 -23969.117,E2 -23969.117} C_VEL
LIN {X 0,Y 156.742,Z 501.539,A -85,B 0,C 180,E1 -23970.666,E2 -23970.666} C_VEL
LIN {X 0,Y 158.906,Z 503.572,A -85,B 0,C 180,E1 -23972.137,E2 -23972.137} C_VEL
LIN {X 0,Y 161.51,Z 507.252,A -85,B 0,C 180,E1 -23973.88,E2 -23973.88} C_VEL
LIN {X 0,Y 162.978,Z 509.115,A -85,B 0,C 180,E1 -23974.788,E2 -23974.788} C_VEL
LIN {X 0,Y 166.411,Z 513.885,A -85,B 0,C 180,E1 -23976.806,E2 -23976.806} C_VEL
LIN {X 0,Y 171.509,Z 521.273,A -85,B 0,C 180,E1 -23979.521,E2 -23979.521} C_VEL
LIN {X 0,Y 177.993,Z 531.767,A -85,B 0,C 180,E1 -23982.622,E2 -23982.622} C_VEL
LIN {X 0,Y 184.072,Z 543.159,A -85,B 0,C 180,E1 -23985.272,E2 -23985.272} C_VEL
LIN {X 0,Y 189.756,Z 555.786,A -85,B 0,C 180,E1 -23987.598,E2 -23987.598} C_VEL
LIN {X 0,Y 196.355,Z 570.897,A -85,B 0,C 180,E1 -23990.056,E2 -23990.056} C_VEL
LIN {X 0,Y 204.632,Z 585.908,A -85,B 0,C 180,E1 -23992.677,E2 -23992.677} C_VEL
LIN {X 0,Y 211.511,Z 596.726,A -85,B 0,C 180,E1 -23994.798,E2 -23994.798} C_VEL
LIN {X 0,Y 218.17,Z 606.024,A -85,B 0,C 180,E1 -23996.876,E2 -23996.876} C_VEL
LIN {X 0,Y 226.054,Z 615.945,A -85,B 0,C 180,E1 -23999.313,E2 -23999.313} C_VEL
LIN {X 0,Y 234.945,Z 625.613,A -85,B 0,C 180,E1 -24001.932,E2 -24001.932} C_VEL
LIN {X 0,Y 246.23,Z 635.81,A -85,B 0,C 180,E1 -24004.98,E2 -24004.98} C_VEL
LIN {X 0,Y 257.971,Z 644.659,A -85,B 0,C 180,E1 -24007.853,E2 -24007.853} C_VEL
LIN {X 0,Y 268.721,Z 651.822,A -85,B 0,C 180,E1 -24010.301,E2 -24010.301} C_VEL
LIN {X 0,Y 279.627,Z 658.8,A -85,B 0,C 180,E1 -24012.75,E2 -24012.75} C_VEL
LIN {X 0,Y 287.841,Z 664.098,A -85,B 0,C 180,E1 -24014.661,E2 -24014.661} C_VEL
LIN {X 0,Y 293.557,Z 668.036,A -85,B 0,C 180,E1 -24016.149,E2 -24016.149} C_VEL
LIN {X 0,Y 299.461,Z 671.891,A -85,B 0,C 180,E1 -24017.806,E2 -24017.806} C_VEL
LIN {X 0,Y 304.101,Z 674.865,A -85,B 0,C 180,E1 -24019.346,E2 -24019.346} C_VEL
LIN {X 0,Y 307.578,Z 677.316,A -85,B 0,C 180,E1 -24020.796,E2 -24020.796} C_VEL
LIN {X 0,Y 311.699,Z 679.876,A -85,B 0,C 180,E1 -24022.765,E2 -24022.765} C_VEL
LIN {X 0,Y 315.277,Z 681.806,A -85,B 0,C 180,E1 -24024.884,E2 -24024.884} C_VEL
LIN {X 0,Y 317.041,Z 682.548,A -85,B 0,C 180,E1 -24026.187,E2 -24026.187} C_VEL
LIN {X 0,Y 318.356,Z 683.048,A -85,B 0,C 180,E1 -24027.469,E2 -24027.469} C_VEL
LIN {X 0,Y 319.06,Z 683.372,A -85,B 0,C 180,E1 -24028.738,E2 -24028.738} C_VEL
LIN {X 0,Y 319.431,Z 683.427,A -85,B 0,C 180,E1 -24030,E2 -24030} C_VEL
LIN {X 0,Y 319.068,Z 683.365,A -85,B 0,C 180,E1 -24031.262,E2 -24031.262} C_VEL
LIN {X 0,Y 318.356,Z 683.046,A -85,B 0,C 180,E1 -24032.531,E2 -24032.531} C_VEL
LIN {X 0,Y 316.971,Z 682.519,A -85,B 0,C 180,E1 -24033.878,E2 -24033.878} C_VEL
LIN {X 0,Y 315.264,Z 681.812,A -85,B 0,C 180,E1 -24035.116,E2 -24035.116} C_VEL
LIN {X 0,Y 311.676,Z 679.929,A -85,B 0,C 180,E1 -24037.201,E2 -24037.201} C_VEL
LIN {X 0,Y 307.556,Z 677.303,A -85,B 0,C 180,E1 -24039.204,E2 -24039.204} C_VEL
LIN {X 0,Y 304.069,Z 674.859,A -85,B 0,C 180,E1 -24040.655,E2 -24040.655} C_VEL
LIN {X 0,Y 299.399,Z 671.87,A -85,B 0,C 180,E1 -24042.196,E2 -24042.196} C_VEL
LIN {X 0,Y 292.278,Z 667.133,A -85,B 0,C 180,E1 -24044.215,E2 -24044.215} C_VEL
LIN {X 0,Y 285.114,Z 662.279,A -85,B 0,C 180,E1 -24045.994,E2 -24045.994} C_VEL
LIN {X 0,Y 274.173,Z 655.237,A -85,B 0,C 180,E1 -24048.489,E2 -24048.489} C_VEL
LIN {X 0,Y 263.325,Z 648.262,A -85,B 0,C 180,E1 -24050.92,E2 -24050.92} C_VEL
LIN {X 0,Y 251.012,Z 639.577,A -85,B 0,C 180,E1 -24053.814,E2 -24053.814} C_VEL
LIN {X 0,Y 240.819,Z 631.1,A -85,B 0,C 180,E1 -24056.45,E2 -24056.45} C_VEL
LIN {X 0,Y 231.69,Z 622.123,A -85,B 0,C 180,E1 -24059.034,E2 -24059.034} C_VEL
LIN {X 0,Y 221.723,Z 610.617,A -85,B 0,C 180,E1 -24062.023,E2 -24062.023} C_VEL
LIN {X 0,Y 213.6,Z 599.738,A -85,B 0,C 180,E1 -24064.55,E2 -24064.55} C_VEL
LIN {X 0,Y 207.535,Z 590.449,A -85,B 0,C 180,E1 -24066.466,E2 -24066.466} C_VEL
LIN {X 0,Y 200.665,Z 579.043,A -85,B 0,C 180,E1 -24068.547,E2 -24068.547} C_VEL
LIN {X 0,Y 193.42,Z 564.629,A -85,B 0,C 180,E1 -24070.983,E2 -24070.983} C_VEL
LIN {X 0,Y 186.355,Z 547.997,A -85,B 0,C 180,E1 -24073.778,E2 -24073.778} C_VEL
LIN {X 0,Y 181.096,Z 537.426,A -85,B 0,C 180,E1 -24075.996,E2 -24075.996} C_VEL
LIN {X 0,Y 175.144,Z 526.984,A -85,B 0,C 180,E1 -24078.699,E2 -24078.699} C_VEL
LIN {X 0,Y 169.933,Z 518.99,A -85,B 0,C 180,E1 -24081.284,E2 -24081.284} C_VEL
LIN {X 0,Y 165.253,Z 512.147,A -85,B 0,C 180,E1 -24083.864,E2 -24083.864} C_VEL
LIN {X 0,Y 162.546,Z 508.374,A -85,B 0,C 180,E1 -24085.49,E2 -24085.49} C_VEL
LIN {X 0,Y 159.39,Z 504.453,A -85,B 0,C 180,E1 -24087.512,E2 -24087.512} C_VEL
LIN {X 0,Y 158.4,Z 503.002,A -85,B 0,C 180,E1 -24088.206,E2 -24088.206} C_VEL
LIN {X 0,Y 155.939,Z 500.486,A -85,B 0,C 180,E1 -24089.935,E2 -24089.935} C_VEL
LIN {X 0,Y 154.515,Z 497.964,A -85,B 0,C 180,E1 -24091.106,E2 -24091.106} C_VEL
LIN {X 0,Y 151.837,Z 495.948,A -85,B 0,C 180,E1 -24093.218,E2 -24093.218} C_VEL
LIN {X 0,Y 150.333,Z 493.071,A -85,B 0,C 180,E1 -24094.865,E2 -24094.865} C_VEL
LIN {X 0,Y 150.212,Z 492.312,A -85,B 0,C 180,E1 -24096.205,E2 -24096.205} C_VEL
LIN {X 0,Y 150.292,Z 492.214,A -85,B 0,C 180,E1 -24100.898,E2 -24100.898} C_VEL
LIN {X 0,Y 150.4,Z 492.227,A -85,B 0,C 180,E1 -24106.493,E2 -24106.493} C_VEL
LIN {X 0,Y 150.601,Z 492.17,A -85,B 0,C 180,E1 -24109.246,E2 -24109.246} C_VEL
LIN {X 0,Y 150.675,Z 492.173,A -85,B 0,C 180,E1 -24111.96,E2 -24111.96} C_VEL
LIN {X 0,Y 151.191,Z 492.094,A -85,B 0,C 180,E1 -24120.004,E2 -24120.004} C_VEL
LIN {X 0,Y 150.676,Z 492.163,A -85,B 0,C 180,E1 -24128.048,E2 -24128.048} C_VEL
LIN {X 0,Y 150.57,Z 492.184,A -85,B 0,C 180,E1 -24131.425,E2 -24131.425} C_VEL
LIN {X 0,Y 150.302,Z 492.222,A -85,B 0,C 180,E1 -24136.297,E2 -24136.297} C_VEL
LIN {X 0,Y 150.283,Z 492.227,A -85,B 0,C 180,E1 -24140.725,E2 -24140.725} C_VEL
LIN {X 0,Y 150.252,Z 492.515,A -85,B 0,C 180,E1 -24144.164,E2 -24144.164} C_VEL
LIN {X 0,Y 150.538,Z 493.716,A -85,B 0,C 180,E1 -24145.107,E2 -24145.107} C_VEL
LIN {X 0,Y 151.987,Z 496.1,A -85,B 0,C 180,E1 -24146.522,E2 -24146.522} C_VEL
LIN {X 0,Y 154.816,Z 498.396,A -85,B 0,C 180,E1 -24148.749,E2 -24148.749} C_VEL
LIN {X 0,Y 156.72,Z 501.489,A -85,B 0,C 180,E1 -24150.259,E2 -24150.259} C_VEL
LIN {X 0,Y 158.941,Z 503.646,A -85,B 0,C 180,E1 -24151.775,E2 -24151.775} C_VEL
LIN {X 0,Y 161.54,Z 507.265,A -85,B 0,C 180,E1 -24153.507,E2 -24153.507} C_VEL
LIN {X 0,Y 162.739,Z 508.758,A -85,B 0,C 180,E1 -24154.25,E2 -24154.25} C_VEL
LIN {X 0,Y 165.786,Z 513.249,A -85,B 0,C 180,E1 -24156.08,E2 -24156.08} C_VEL
LIN {X 0,Y 170.648,Z 521.617,A -85,B 0,C 180,E1 -24158.8,E2 -24158.8} C_VEL
LIN {X 0,Y 177.433,Z 535.163,A -85,B 0,C 180,E1 -24162.235,E2 -24162.235} C_VEL
LIN {X 0,Y 182.632,Z 547.693,A -85,B 0,C 180,E1 -24164.678,E2 -24164.678} C_VEL
LIN {X 0,Y 184.727,Z 553.722,A -85,B 0,C 180,E1 -24165.648,E2 -24165.648} C_VEL
LIN {X 0,Y 185.371,Z 559.614,A -85,B 0,C 180,E1 -24166.151,E2 -24166.151} C_VEL
LIN {X 0,Y 182.972,Z 596.729,A -85,B 0,C 180,E1 -24167.48,E2 -24167.48} C_VEL
LIN {X 0,Y 181.683,Z 607.143,A -85,B 0,C 180,E1 -24168.066,E2 -24168.066} C_VEL
LIN {X 0,Y 179.985,Z 616.522,A -85,B 0,C 180,E1 -24168.782,E2 -24168.782} C_VEL
LIN {X 0,Y 177.956,Z 625.613,A -85,B 0,C 180,E1 -24169.708,E2 -24169.708} C_VEL
LIN {X 0,Y 175.489,Z 634.755,A -85,B 0,C 180,E1 -24170.895,E2 -24170.895} C_VEL
LIN {X 0,Y 172.623,Z 643.752,A -85,B 0,C 180,E1 -24172.361,E2 -24172.361} C_VEL
LIN {X 0,Y 169.52,Z 652.476,A -85,B 0,C 180,E1 -24174.155,E2 -24174.155} C_VEL
LIN {X 0,Y 166.521,Z 659.892,A -85,B 0,C 180,E1 -24175.999,E2 -24175.999} C_VEL
LIN {X 0,Y 162.634,Z 668.684,A -85,B 0,C 180,E1 -24178.765,E2 -24178.765} C_VEL
LIN {X 0,Y 159.923,Z 674.675,A -85,B 0,C 180,E1 -24181.092,E2 -24181.092} C_VEL
LIN {X 0,Y 156.94,Z 680.989,A -85,B 0,C 180,E1 -24184.112,E2 -24184.112} C_VEL
LIN {X 0,Y 154.182,Z 686.26,A -85,B 0,C 180,E1 -24187.204,E2 -24187.204} C_VEL
LIN {X 0,Y 151.553,Z 691.356,A -85,B 0,C 180,E1 -24191.058,E2 -24191.058} C_VEL
LIN {X 0,Y 149.632,Z 695.324,A -85,B 0,C 180,E1 -24195.029,E2 -24195.029} C_VEL
LIN {X 0,Y 148.394,Z 698.267,A -85,B 0,C 180,E1 -24199.08,E2 -24199.08} C_VEL
LIN {X 0,Y 147.88,Z 699.772,A -85,B 0,C 180,E1 -24201.803,E2 -24201.803} C_VEL
LIN {X 0,Y 147.576,Z 701.309,A -85,B 0,C 180,E1 -24207.27,E2 -24207.27} C_VEL
LIN {X 0,Y 147.685,Z 701.593,A -85,B 0,C 180,E1 -24210,E2 -24210} C_VEL
LIN {X 0,Y 147.63,Z 700.707,A -85,B 0,C 180,E1 -24215.463,E2 -24215.463} C_VEL
LIN {X 0,Y 147.891,Z 699.773,A -85,B 0,C 180,E1 -24218.196,E2 -24218.196} C_VEL
LIN {X 0,Y 149.143,Z 696.415,A -85,B 0,C 180,E1 -24223.628,E2 -24223.628} C_VEL
LIN {X 0,Y 150.82,Z 692.784,A -85,B 0,C 180,E1 -24227.631,E2 -24227.631} C_VEL
LIN {X 0,Y 153.27,Z 688.052,A -85,B 0,C 180,E1 -24231.52,E2 -24231.52} C_VEL
LIN {X 0,Y 156.383,Z 682.082,A -85,B 0,C 180,E1 -24235.273,E2 -24235.273} C_VEL
LIN {X 0,Y 159.207,Z 676.234,A -85,B 0,C 180,E1 -24238.195,E2 -24238.195} C_VEL
LIN {X 0,Y 161.954,Z 670.246,A -85,B 0,C 180,E1 -24240.656,E2 -24240.656} C_VEL
LIN {X 0,Y 164.956,Z 663.592,A -85,B 0,C 180,E1 -24242.903,E2 -24242.903} C_VEL
LIN {X 0,Y 166.371,Z 660.272,A -85,B 0,C 180,E1 -24243.886,E2 -24243.886} C_VEL
LIN {X 0,Y 167.614,Z 655.936,A -85,B 0,C 180,E1 -24245.201,E2 -24245.201} C_VEL
LIN {X 0,Y 168.121,Z 648.531,A -85,B 0,C 180,E1 -24247.453,E2 -24247.453} C_VEL
LIN {X 0,Y 168.627,Z 640.723,A -85,B 0,C 180,E1 -24249.509,E2 -24249.509} C_VEL
LIN {X 0,Y 169.733,Z 635.593,A -85,B 0,C 180,E1 -24250.449,E2 -24250.449} C_VEL
LIN {X 0,Y 172.046,Z 627.383,A -85,B 0,C 180,E1 -24251.59,E2 -24251.59} C_VEL
LIN {X 0,Y 174.407,Z 617.586,A -85,B 0,C 180,E1 -24252.647,E2 -24252.647} C_VEL
LIN {X 0,Y 176.383,Z 607.504,A -85,B 0,C 180,E1 -24253.436,E2 -24253.436} C_VEL
LIN {X 0,Y 177.734,Z 597.299,A -85,B 0,C 180,E1 -24254.021,E2 -24254.021} C_VEL
LIN {X 0,Y 179.814,Z 567.358,A -85,B 0,C 180,E1 -24255.133,E2 -24255.133} C_VEL
LIN {X 0,Y 180.234,Z 559.805,A -85,B 0,C 180,E1 -24255.417,E2 -24255.417} C_VEL
LIN {X 0,Y 179.604,Z 555.541,A -85,B 0,C 180,E1 -24255.859,E2 -24255.859} C_VEL
LIN {X 0,Y 174.563,Z 542.391,A -85,B 0,C 180,E1 -24258.367,E2 -24258.367} C_VEL
LIN {X 0,Y 168.548,Z 529.622,A -85,B 0,C 180,E1 -24261.552,E2 -24261.552} C_VEL
LIN {X 0,Y 163.885,Z 520.985,A -85,B 0,C 180,E1 -24264.266,E2 -24264.266} C_VEL
LIN {X 0,Y 161.455,Z 516.918,A -85,B 0,C 180,E1 -24265.786,E2 -24265.786} C_VEL
LIN {X 0,Y 158.905,Z 513.28,A -85,B 0,C 180,E1 -24267.449,E2 -24267.449} C_VEL
LIN {X 0,Y 155.77,Z 509.066,A -85,B 0,C 180,E1 -24269.661,E2 -24269.661} C_VEL
LIN {X 0,Y 153.177,Z 506.007,A -85,B 0,C 180,E1 -24271.64,E2 -24271.64} C_VEL
LIN {X 0,Y 152.189,Z 504.372,A -85,B 0,C 180,E1 -24272.493,E2 -24272.493} C_VEL
LIN {X 0,Y 149.46,Z 501.883,A -85,B 0,C 180,E1 -24274.829,E2 -24274.829} C_VEL
LIN {X 0,Y 147.834,Z 498.991,A -85,B 0,C 180,E1 -24276.533,E2 -24276.533} C_VEL
LIN {X 0,Y 145.25,Z 497.246,A -85,B 0,C 180,E1 -24279.214,E2 -24279.214} C_VEL
LIN {X 0,Y 143.597,Z 494.642,A -85,B 0,C 180,E1 -24281.446,E2 -24281.446} C_VEL
LIN {X 0,Y 143.294,Z 493.558,A -85,B 0,C 180,E1 -24282.514,E2 -24282.514} C_VEL
LIN {X 0,Y 143.278,Z 493.149,A -85,B 0,C 180,E1 -24284.344,E2 -24284.344} C_VEL
LIN {X 0,Y 143.528,Z 493.058,A -85,B 0,C 180,E1 -24288.701,E2 -24288.701} C_VEL
LIN {X 0,Y 143.602,Z 493.04,A -85,B 0,C 180,E1 -24291.553,E2 -24291.553} C_VEL
LIN {X 0,Y 144.149,Z 492.97,A -85,B 0,C 180,E1 -24299.996,E2 -24299.996} C_VEL
LIN {X 0,Y 143.601,Z 493.048,A -85,B 0,C 180,E1 -24308.438,E2 -24308.438} C_VEL
LIN {X 0,Y 143.493,Z 493.06,A -85,B 0,C 180,E1 -24311.608,E2 -24311.608} C_VEL
LIN {X 0,Y 143.258,Z 493.407,A -85,B 0,C 180,E1 -24317.574,E2 -24317.574} C_VEL
LIN {X 0,Y 143.589,Z 494.568,A -85,B 0,C 180,E1 -24318.916,E2 -24318.916} C_VEL
LIN {X 0,Y 145.121,Z 497.141,A -85,B 0,C 180,E1 -24321.027,E2 -24321.027} C_VEL
LIN {X 0,Y 148.045,Z 499.255,A -85,B 0,C 180,E1 -24324.072,E2 -24324.072} C_VEL
LIN {X 0,Y 149.805,Z 502.295,A -85,B 0,C 180,E1 -24325.881,E2 -24325.881} C_VEL
LIN {X 0,Y 152.529,Z 504.778,A -85,B 0,C 180,E1 -24328.178,E2 -24328.178} C_VEL
LIN {X 0,Y 154.719,Z 508.095,A -85,B 0,C 180,E1 -24329.973,E2 -24329.973} C_VEL
LIN {X 0,Y 156.483,Z 509.923,A -85,B 0,C 180,E1 -24331.243,E2 -24331.243} C_VEL
LIN {X 0,Y 159.388,Z 513.83,A -85,B 0,C 180,E1 -24333.253,E2 -24333.253} C_VEL
LIN {X 0,Y 163.894,Z 520.356,A -85,B 0,C 180,E1 -24336.081,E2 -24336.081} C_VEL
LIN {X 0,Y 170.021,Z 529.636,A -85,B 0,C 180,E1 -24339.455,E2 -24339.455} C_VEL
LIN {X 0,Y 175.642,Z 539.423,A -85,B 0,C 180,E1 -24342.236,E2 -24342.236} C_VEL
LIN {X 0,Y 180.928,Z 549.977,A -85,B 0,C 180,E1 -24344.65,E2 -24344.65} C_VEL
LIN {X 0,Y 185.886,Z 561.637,A -85,B 0,C 180,E1 -24346.797,E2 -24346.797} C_VEL
LIN {X 0,Y 192.225,Z 576.155,A -85,B 0,C 180,E1 -24349.265,E2 -24349.265} C_VEL
LIN {X 0,Y 199.559,Z 589.859,A -85,B 0,C 180,E1 -24351.788,E2 -24351.788} C_VEL
LIN {X 0,Y 206.554,Z 601.352,A -85,B 0,C 180,E1 -24354.215,E2 -24354.215} C_VEL
LIN {X 0,Y 214.487,Z 612.666,A -85,B 0,C 180,E1 -24356.972,E2 -24356.972} C_VEL
LIN {X 0,Y 223.308,Z 623.478,A -85,B 0,C 180,E1 -24359.93,E2 -24359.93} C_VEL
LIN {X 0,Y 232.862,Z 633.381,A -85,B 0,C 180,E1 -24362.91,E2 -24362.91} C_VEL
LIN {X 0,Y 242.86,Z 641.961,A -85,B 0,C 180,E1 -24365.735,E2 -24365.735} C_VEL
LIN {X 0,Y 256.261,Z 651.389,A -85,B 0,C 180,E1 -24369.113,E2 -24369.113} C_VEL
LIN {X 0,Y 269.42,Z 659.526,A -85,B 0,C 180,E1 -24372.187,E2 -24372.187} C_VEL
LIN {X 0,Y 280.382,Z 666.191,A -85,B 0,C 180,E1 -24374.792,E2 -24374.792} C_VEL
LIN {X 0,Y 285.854,Z 669.644,A -85,B 0,C 180,E1 -24376.188,E2 -24376.188} C_VEL
LIN {X 0,Y 291.636,Z 673.412,A -85,B 0,C 180,E1 -24377.788,E2 -24377.788} C_VEL
LIN {X 0,Y 295.726,Z 675.981,A -85,B 0,C 180,E1 -24379.04,E2 -24379.04} C_VEL
LIN {X 0,Y 299.356,Z 678.462,A -85,B 0,C 180,E1 -24380.397,E2 -24380.397} C_VEL
LIN {X 0,Y 304.61,Z 681.895,A -85,B 0,C 180,E1 -24382.771,E2 -24382.771} C_VEL
LIN {X 0,Y 308.104,Z 683.814,A -85,B 0,C 180,E1 -24384.765,E2 -24384.765} C_VEL
LIN {X 0,Y 310.043,Z 684.716,A -85,B 0,C 180,E1 -24386.101,E2 -24386.101} C_VEL
LIN {X 0,Y 311.465,Z 685.277,A -85,B 0,C 180,E1 -24387.413,E2 -24387.413} C_VEL
LIN {X 0,Y 312.282,Z 685.61,A -85,B 0,C 180,E1 -24388.71,E2 -24388.71} C_VEL
LIN {X 0,Y 312.7,Z 685.677,A -85,B 0,C 180,E1 -24390,E2 -24390} C_VEL
LIN {X 0,Y 312.288,Z 685.61,A -85,B 0,C 180,E1 -24391.29,E2 -24391.29} C_VEL
LIN {X 0,Y 311.466,Z 685.281,A -85,B 0,C 180,E1 -24392.587,E2 -24392.587} C_VEL
LIN {X 0,Y 309.959,Z 684.69,A -85,B 0,C 180,E1 -24393.966,E2 -24393.966} C_VEL
LIN {X 0,Y 308.084,Z 683.84,A -85,B 0,C 180,E1 -24395.235,E2 -24395.235} C_VEL
LIN {X 0,Y 304.587,Z 681.944,A -85,B 0,C 180,E1 -24397.194,E2 -24397.194} C_VEL
LIN {X 0,Y 301.407,Z 679.873,A -85,B 0,C 180,E1 -24398.717,E2 -24398.717} C_VEL
LIN {X 0,Y 297.931,Z 677.493,A -85,B 0,C 180,E1 -24400.19,E2 -24400.19} C_VEL
LIN {X 0,Y 294.028,Z 674.926,A -85,B 0,C 180,E1 -24401.492,E2 -24401.492} C_VEL
LIN {X 0,Y 288.567,Z 671.448,A -85,B 0,C 180,E1 -24403.058,E2 -24403.058} C_VEL
LIN {X 0,Y 280.398,Z 666.145,A -85,B 0,C 180,E1 -24405.22,E2 -24405.22} C_VEL
LIN {X 0,Y 269.422,Z 659.519,A -85,B 0,C 180,E1 -24407.814,E2 -24407.814} C_VEL
LIN {X 0,Y 254.015,Z 649.894,A -85,B 0,C 180,E1 -24411.441,E2 -24411.441} C_VEL
LIN {X 0,Y 241.945,Z 641.2,A -85,B 0,C 180,E1 -24414.515,E2 -24414.515} C_VEL
LIN {X 0,Y 230.399,Z 631.088,A -85,B 0,C 180,E1 -24417.805,E2 -24417.805} C_VEL
LIN {X 0,Y 220.972,Z 620.773,A -85,B 0,C 180,E1 -24420.832,E2 -24420.832} C_VEL
LIN {X 0,Y 213.124,Z 610.831,A -85,B 0,C 180,E1 -24423.486,E2 -24423.486} C_VEL
LIN {X 0,Y 205.832,Z 600.262,A -85,B 0,C 180,E1 -24426.028,E2 -24426.028} C_VEL
LIN {X 0,Y 198.734,Z 588.338,A -85,B 0,C 180,E1 -24428.523,E2 -24428.523} C_VEL
LIN {X 0,Y 190.934,Z 573.521,A -85,B 0,C 180,E1 -24431.201,E2 -24431.201} C_VEL
LIN {X 0,Y 181.975,Z 552.331,A -85,B 0,C 180,E1 -24434.886,E2 -24434.886} C_VEL
LIN {X 0,Y 177.054,Z 542.121,A -85,B 0,C 180,E1 -24437.101,E2 -24437.101} C_VEL
LIN {X 0,Y 171.593,Z 532.295,A -85,B 0,C 180,E1 -24439.738,E2 -24439.738} C_VEL
LIN {X 0,Y 166.46,Z 524.15,A -85,B 0,C 180,E1 -24442.451,E2 -24442.451} C_VEL
LIN {X 0,Y 161.805,Z 517.381,A -85,B 0,C 180,E1 -24445.181,E2 -24445.181} C_VEL
LIN {X 0,Y 158.956,Z 513.385,A -85,B 0,C 180,E1 -24447.023,E2 -24447.023} C_VEL
LIN {X 0,Y 155.822,Z 509.143,A -85,B 0,C 180,E1 -24449.232,E2 -24449.232} C_VEL
LIN {X 0,Y 153.31,Z 506.235,A -85,B 0,C 180,E1 -24451.138,E2 -24451.138} C_VEL
LIN {X 0,Y 152.162,Z 504.383,A -85,B 0,C 180,E1 -24452.123,E2 -24452.123} C_VEL
LIN {X 0,Y 149.455,Z 501.864,A -85,B 0,C 180,E1 -24454.446,E2 -24454.446} C_VEL
LIN {X 0,Y 147.808,Z 499.001,A -85,B 0,C 180,E1 -24456.166,E2 -24456.166} C_VEL
LIN {X 0,Y 145.121,Z 497.141,A -85,B 0,C 180,E1 -24458.973,E2 -24458.973} C_VEL
LIN {X 0,Y 143.543,Z 494.424,A -85,B 0,C 180,E1 -24461.17,E2 -24461.17} C_VEL
LIN {X 0,Y 143.26,Z 493.387,A -85,B 0,C 180,E1 -24462.518,E2 -24462.518} C_VEL
LIN {X 0,Y 143.528,Z 493.053,A -85,B 0,C 180,E1 -24468.709,E2 -24468.709} C_VEL
LIN {X 0,Y 143.601,Z 493.048,A -85,B 0,C 180,E1 -24471.562,E2 -24471.562} C_VEL
LIN {X 0,Y 144.149,Z 492.97,A -85,B 0,C 180,E1 -24480.004,E2 -24480.004} C_VEL
LIN {X 0,Y 143.602,Z 493.04,A -85,B 0,C 180,E1 -24488.447,E2 -24488.447} C_VEL
LIN {X 0,Y 143.493,Z 493.066,A -85,B 0,C 180,E1 -24491.608,E2 -24491.608} C_VEL
LIN {X 0,Y 143.272,Z 493.405,A -85,B 0,C 180,E1 -24497.213,E2 -24497.213} C_VEL
LIN {X 0,Y 143.555,Z 494.478,A -85,B 0,C 180,E1 -24498.467,E2 -24498.467} C_VEL
LIN {X 0,Y 145.078,Z 497.055,A -85,B 0,C 180,E1 -24500.581,E2 -24500.581} C_VEL
LIN {X 0,Y 147.5,Z 498.848,A -85,B 0,C 180,E1 -24503.151,E2 -24503.151} C_VEL
LIN {X 0,Y 148.138,Z 499.446,A -85,B 0,C 180,E1 -24503.786,E2 -24503.786} C_VEL
LIN {X 0,Y 149.696,Z 502.143,A -85,B 0,C 180,E1 -24505.389,E2 -24505.389} C_VEL
LIN {X 0,Y 152.546,Z 504.867,A -85,B 0,C 180,E1 -24507.81,E2 -24507.81} C_VEL
LIN {X 0,Y 155.139,Z 508.525,A -85,B 0,C 180,E1 -24509.893,E2 -24509.893} C_VEL
LIN {X 0,Y 156.573,Z 510.09,A -85,B 0,C 180,E1 -24510.923,E2 -24510.923} C_VEL
LIN {X 0,Y 160.296,Z 515.249,A -85,B 0,C 180,E1 -24513.472,E2 -24513.472} C_VEL
LIN {X 0,Y 162.748,Z 518.978,A -85,B 0,C 180,E1 -24515.028,E2 -24515.028} C_VEL
LIN {X 0,Y 167.074,Z 526.667,A -85,B 0,C 180,E1 -24517.609,E2 -24517.609} C_VEL
LIN {X 0,Y 173.605,Z 540.133,A -85,B 0,C 180,E1 -24521.14,E2 -24521.14} C_VEL
LIN {X 0,Y 179.035,Z 553.912,A -85,B 0,C 180,E1 -24523.863,E2 -24523.863} C_VEL
LIN {X 0,Y 179.999,Z 557.562,A -85,B 0,C 180,E1 -24524.383,E2 -24524.383} C_VEL
LIN {X 0,Y 180.195,Z 561.228,A -85,B 0,C 180,E1 -24524.649,E2 -24524.649} C_VEL
LIN {X 0,Y 177.812,Z 596.333,A -85,B 0,C 180,E1 -24525.92,E2 -24525.92} C_VEL
LIN {X 0,Y 176.525,Z 606.633,A -85,B 0,C 180,E1 -24526.508,E2 -24526.508} C_VEL
LIN {X 0,Y 174.72,Z 616.326,A -85,B 0,C 180,E1 -24527.252,E2 -24527.252} C_VEL
LIN {X 0,Y 172.602,Z 625.417,A -85,B 0,C 180,E1 -24528.183,E2 -24528.183} C_VEL
LIN {X 0,Y 170.052,Z 634.559,A -85,B 0,C 180,E1 -24529.389,E2 -24529.389} C_VEL
LIN {X 0,Y 167.049,Z 643.555,A -85,B 0,C 180,E1 -24530.871,E2 -24530.871} C_VEL
LIN {X 0,Y 163.824,Z 652.28,A -85,B 0,C 180,E1 -24532.703,E2 -24532.703} C_VEL
LIN {X 0,Y 160.681,Z 659.696,A -85,B 0,C 180,E1 -24534.582,E2 -24534.582} C_VEL
LIN {X 0,Y 156.592,Z 668.487,A -85,B 0,C 180,E1 -24537.414,E2 -24537.414} C_VEL
LIN {X 0,Y 153.718,Z 674.478,A -85,B 0,C 180,E1 -24539.807,E2 -24539.807} C_VEL
LIN {X 0,Y 150.552,Z 680.792,A -85,B 0,C 180,E1 -24542.926,E2 -24542.926} C_VEL
LIN {X 0,Y 147.631,Z 686.063,A -85,B 0,C 180,E1 -24546.131,E2 -24546.131} C_VEL
LIN {X 0,Y 144.818,Z 691.158,A -85,B 0,C 180,E1 -24550.141,E2 -24550.141} C_VEL
LIN {X 0,Y 142.734,Z 695.127,A -85,B 0,C 180,E1 -24554.288,E2 -24554.288} C_VEL
LIN {X 0,Y 141.405,Z 698.07,A -85,B 0,C 180,E1 -24558.533,E2 -24558.533} C_VEL
LIN {X 0,Y 140.837,Z 699.576,A -85,B 0,C 180,E1 -24561.39,E2 -24561.39} C_VEL
LIN {X 0,Y 140.494,Z 701.113,A -85,B 0,C 180,E1 -24567.133,E2 -24567.133} C_VEL
LIN {X 0,Y 140.571,Z 701.386,A -85,B 0,C 180,E1 -24570.29,E2 -24570.29} C_VEL
LIN {X 0,Y 140.554,Z 700.51,A -85,B 0,C 180,E1 -24575.739,E2 -24575.739} C_VEL
LIN {X 0,Y 140.845,Z 699.576,A -85,B 0,C 180,E1 -24578.609,E2 -24578.609} C_VEL
LIN {X 0,Y 142.226,Z 696.219,A -85,B 0,C 180,E1 -24584.304,E2 -24584.304} C_VEL
LIN {X 0,Y 144.031,Z 692.587,A -85,B 0,C 180,E1 -24588.491,E2 -24588.491} C_VEL
LIN {X 0,Y 146.639,Z 687.854,A -85,B 0,C 180,E1 -24592.545,E2 -24592.545} C_VEL
LIN {X 0,Y 149.951,Z 681.884,A -85,B 0,C 180,E1 -24596.439,E2 -24596.439} C_VEL
LIN {X 0,Y 152.777,Z 676.366,A -85,B 0,C 180,E1 -24599.306,E2 -24599.306} C_VEL
LIN {X 0,Y 155.859,Z 670.048,A -85,B 0,C 180,E1 -24601.994,E2 -24601.994} C_VEL
LIN {X 0,Y 159.037,Z 663.396,A -85,B 0,C 180,E1 -24604.293,E2 -24604.293} C_VEL
LIN {X 0,Y 162.417,Z 655.571,A -85,B 0,C 180,E1 -24606.511,E2 -24606.511} C_VEL
LIN {X 0,Y 165.688,Z 647.494,A -85,B 0,C 180,E1 -24608.341,E2 -24608.341} C_VEL
LIN {X 0,Y 169.043,Z 637.737,A -85,B 0,C 180,E1 -24610.121,E2 -24610.121} C_VEL
LIN {X 0,Y 169.733,Z 635.593,A -85,B 0,C 180,E1 -24610.449,E2 -24610.449} C_VEL
LIN {X 0,Y 170.779,Z 630.471,A -85,B 0,C 180,E1 -24611.349,E2 -24611.349} C_VEL
LIN {X 0,Y 170.831,Z 621.853,A -85,B 0,C 180,E1 -24613.049,E2 -24613.049} C_VEL
LIN {X 0,Y 170.719,Z 612.999,A -85,B 0,C 180,E1 -24614.525,E2 -24614.525} C_VEL
LIN {X 0,Y 171.292,Z 607.37,A -85,B 0,C 180,E1 -24615.063,E2 -24615.063} C_VEL
LIN {X 0,Y 172.628,Z 597.883,A -85,B 0,C 180,E1 -24615.621,E2 -24615.621} C_VEL
LIN {X 0,Y 174.364,Z 574.831,A -85,B 0,C 180,E1 -24616.511,E2 -24616.511} C_VEL
LIN {X 0,Y 175.243,Z 561.047,A -85,B 0,C 180,E1 -24617.014,E2 -24617.014} C_VEL
LIN {X 0,Y 174.636,Z 557.82,A -85,B 0,C 180,E1 -24617.418,E2 -24617.418} C_VEL
LIN {X 0,Y 169.46,Z 544.309,A -85,B 0,C 180,E1 -24620.209,E2 -24620.209} C_VEL
LIN {X 0,Y 163.404,Z 531.369,A -85,B 0,C 180,E1 -24623.74,E2 -24623.74} C_VEL
LIN {X 0,Y 158.791,Z 522.929,A -85,B 0,C 180,E1 -24626.73,E2 -24626.73} C_VEL
LIN {X 0,Y 155.835,Z 518.742,A -85,B 0,C 180,E1 -24628.772,E2 -24628.772} C_VEL
LIN {X 0,Y 153.33,Z 515.253,A -85,B 0,C 180,E1 -24630.663,E2 -24630.663} C_VEL
LIN {X 0,Y 150.546,Z 511.612,A -85,B 0,C 180,E1 -24632.96,E2 -24632.96} C_VEL
LIN {X 0,Y 149.488,Z 510.4,A -85,B 0,C 180,E1 -24633.887,E2 -24633.887} C_VEL
LIN {X 0,Y 146.818,Z 507.228,A -85,B 0,C 180,E1 -24636.455,E2 -24636.455} C_VEL
LIN {X 0,Y 146.038,Z 505.682,A -85,B 0,C 180,E1 -24637.352,E2 -24637.352} C_VEL
LIN {X 0,Y 143.528,Z 503.744,A -85,B 0,C 180,E1 -24640.137,E2 -24640.137} C_VEL
LIN {X 0,Y 141.703,Z 500.629,A -85,B 0,C 180,E1 -24642.776,E2 -24642.776} C_VEL
LIN {X 0,Y 140.845,Z 499.843,A -85,B 0,C 180,E1 -24644.067,E2 -24644.067} C_VEL
LIN {X 0,Y 138.376,Z 497.971,A -85,B 0,C 180,E1 -24648.557,E2 -24648.557} C_VEL
LIN {X 0,Y 136.7,Z 494.746,A -85,B 0,C 180,E1 -24654.834,E2 -24654.834} C_VEL
LIN {X 0,Y 137.106,Z 493.989,A -85,B 0,C 180,E1 -24659.996,E2 -24659.996} C_VEL
LIN {X 0,Y 136.693,Z 494.763,A -85,B 0,C 180,E1 -24665.527,E2 -24665.527} C_VEL
LIN {X 0,Y 139.74,Z 499.277,A -85,B 0,C 180,E1 -24674.56,E2 -24674.56} C_VEL
LIN {X 0,Y 141.64,Z 500.456,A -85,B 0,C 180,E1 -24677.502,E2 -24677.502} C_VEL
LIN {X 0,Y 143.376,Z 503.593,A -85,B 0,C 180,E1 -24680.063,E2 -24680.063} C_VEL
LIN {X 0,Y 145.696,Z 505.516,A -85,B 0,C 180,E1 -24682.695,E2 -24682.695} C_VEL
LIN {X 0,Y 146.295,Z 506.242,A -85,B 0,C 180,E1 -24683.344,E2 -24683.344} C_VEL
LIN {X 0,Y 148.718,Z 509.722,A -85,B 0,C 180,E1 -24685.821,E2 -24685.821} C_VEL
LIN {X 0,Y 150.376,Z 511.288,A -85,B 0,C 180,E1 -24687.27,E2 -24687.27} C_VEL
LIN {X 0,Y 152.964,Z 514.909,A -85,B 0,C 180,E1 -24689.451,E2 -24689.451} C_VEL
LIN {X 0,Y 154.174,Z 516.344,A -85,B 0,C 180,E1 -24690.374,E2 -24690.374} C_VEL
LIN {X 0,Y 158.076,Z 521.939,A -85,B 0,C 180,E1 -24693.184,E2 -24693.184} C_VEL
LIN {X 0,Y 162.543,Z 528.479,A -85,B 0,C 180,E1 -24696.023,E2 -24696.023} C_VEL
LIN {X 0,Y 168.629,Z 538.46,A -85,B 0,C 180,E1 -24699.458,E2 -24699.458} C_VEL
LIN {X 0,Y 174.684,Z 549.994,A -85,B 0,C 180,E1 -24702.522,E2 -24702.522} C_VEL
LIN {X 0,Y 179.861,Z 561.903,A -85,B 0,C 180,E1 -24704.968,E2 -24704.968} C_VEL
LIN {X 0,Y 187.046,Z 579.189,A -85,B 0,C 180,E1 -24708.029,E2 -24708.029} C_VEL
LIN {X 0,Y 193.833,Z 592.514,A -85,B 0,C 180,E1 -24710.596,E2 -24710.596} C_VEL
LIN {X 0,Y 201.417,Z 605.831,A -85,B 0,C 180,E1 -24713.618,E2 -24713.618} C_VEL
LIN {X 0,Y 208.638,Z 616.415,A -85,B 0,C 180,E1 -24716.42,E2 -24716.42} C_VEL
LIN {X 0,Y 216.481,Z 626.481,A -85,B 0,C 180,E1 -24719.345,E2 -24719.345} C_VEL
LIN {X 0,Y 225.756,Z 636.361,A -85,B 0,C 180,E1 -24722.518,E2 -24722.518} C_VEL
LIN {X 0,Y 235.529,Z 644.859,A -85,B 0,C 180,E1 -24725.508,E2 -24725.508} C_VEL
LIN {X 0,Y 246.704,Z 652.852,A -85,B 0,C 180,E1 -24728.551,E2 -24728.551} C_VEL
LIN {X 0,Y 259.175,Z 660.452,A -85,B 0,C 180,E1 -24731.629,E2 -24731.629} C_VEL
LIN {X 0,Y 270.134,Z 666.718,A -85,B 0,C 180,E1 -24734.273,E2 -24734.273} C_VEL
LIN {X 0,Y 278.178,Z 671.322,A -85,B 0,C 180,E1 -24736.296,E2 -24736.296} C_VEL
LIN {X 0,Y 286.712,Z 676.423,A -85,B 0,C 180,E1 -24738.691,E2 -24738.691} C_VEL
LIN {X 0,Y 291.61,Z 679.467,A -85,B 0,C 180,E1 -24740.288,E2 -24740.288} C_VEL
LIN {X 0,Y 295.134,Z 681.936,A -85,B 0,C 180,E1 -24741.786,E2 -24741.786} C_VEL
LIN {X 0,Y 298.23,Z 683.881,A -85,B 0,C 180,E1 -24743.233,E2 -24743.233} C_VEL
LIN {X 0,Y 300.692,Z 685.241,A -85,B 0,C 180,E1 -24744.636,E2 -24744.636} C_VEL
LIN {X 0,Y 302.903,Z 686.293,A -85,B 0,C 180,E1 -24746.066,E2 -24746.066} C_VEL
LIN {X 0,Y 304.394,Z 686.968,A -85,B 0,C 180,E1 -24747.353,E2 -24747.353} C_VEL
LIN {X 0,Y 305.359,Z 687.36,A -85,B 0,C 180,E1 -24748.681,E2 -24748.681} C_VEL
LIN {X 0,Y 305.838,Z 687.446,A -85,B 0,C 180,E1 -24750,E2 -24750} C_VEL
LIN {X 0,Y 305.364,Z 687.362,A -85,B 0,C 180,E1 -24751.319,E2 -24751.319} C_VEL
LIN {X 0,Y 304.415,Z 686.973,A -85,B 0,C 180,E1 -24752.646,E2 -24752.646} C_VEL
LIN {X 0,Y 302.801,Z 686.28,A -85,B 0,C 180,E1 -24753.993,E2 -24753.993} C_VEL
LIN {X 0,Y 300.657,Z 685.278,A -85,B 0,C 180,E1 -24755.365,E2 -24755.365} C_VEL
LIN {X 0,Y 297.442,Z 683.483,A -85,B 0,C 180,E1 -24757.1,E2 -24757.1} C_VEL
LIN {X 0,Y 293.685,Z 680.944,A -85,B 0,C 180,E1 -24758.844,E2 -24758.844} C_VEL
LIN {X 0,Y 291.558,Z 679.471,A -85,B 0,C 180,E1 -24759.714,E2 -24759.714} C_VEL
LIN {X 0,Y 286.642,Z 676.425,A -85,B 0,C 180,E1 -24761.312,E2 -24761.312} C_VEL
LIN {X 0,Y 280.692,Z 672.832,A -85,B 0,C 180,E1 -24763.023,E2 -24763.023} C_VEL
LIN {X 0,Y 273.642,Z 668.655,A -85,B 0,C 180,E1 -24764.882,E2 -24764.882} C_VEL
LIN {X 0,Y 262.817,Z 662.528,A -85,B 0,C 180,E1 -24767.507,E2 -24767.507} C_VEL
LIN {X 0,Y 250.411,Z 655.132,A -85,B 0,C 180,E1 -24770.52,E2 -24770.52} C_VEL
LIN {X 0,Y 239.643,Z 647.939,A -85,B 0,C 180,E1 -24773.335,E2 -24773.335} C_VEL
LIN {X 0,Y 230.038,Z 640.239,A -85,B 0,C 180,E1 -24776.141,E2 -24776.141} C_VEL
LIN {X 0,Y 221.778,Z 632.316,A -85,B 0,C 180,E1 -24778.819,E2 -24778.819} C_VEL
LIN {X 0,Y 212.023,Z 620.93,A -85,B 0,C 180,E1 -24782.305,E2 -24782.305} C_VEL
LIN {X 0,Y 204.332,Z 610.282,A -85,B 0,C 180,E1 -24785.233,E2 -24785.233} C_VEL
LIN {X 0,Y 198.278,Z 600.464,A -85,B 0,C 180,E1 -24787.635,E2 -24787.635} C_VEL
LIN {X 0,Y 192.457,Z 589.909,A -85,B 0,C 180,E1 -24789.933,E2 -24789.933} C_VEL
LIN {X 0,Y 185.964,Z 576.868,A -85,B 0,C 180,E1 -24792.393,E2 -24792.393} C_VEL
LIN {X 0,Y 177.407,Z 556.004,A -85,B 0,C 180,E1 -24796.174,E2 -24796.174} C_VEL
LIN {X 0,Y 172.544,Z 545.729,A -85,B 0,C 180,E1 -24798.527,E2 -24798.527} C_VEL
LIN {X 0,Y 167.207,Z 536.104,A -85,B 0,C 180,E1 -24801.301,E2 -24801.301} C_VEL
LIN {X 0,Y 161.895,Z 527.431,A -85,B 0,C 180,E1 -24804.375,E2 -24804.375} C_VEL
LIN {X 0,Y 156.256,Z 519.284,A -85,B 0,C 180,E1 -24808.085,E2 -24808.085} C_VEL
LIN {X 0,Y 153.305,Z 515.247,A -85,B 0,C 180,E1 -24810.291,E2 -24810.291} C_VEL
LIN {X 0,Y 150.636,Z 511.778,A -85,B 0,C 180,E1 -24812.488,E2 -24812.488} C_VEL
LIN {X 0,Y 149.955,Z 510.754,A -85,B 0,C 180,E1 -24813.103,E2 -24813.103} C_VEL
LIN {X 0,Y 147.371,Z 508.084,A -85,B 0,C 180,E1 -24815.483,E2 -24815.483} C_VEL
LIN {X 0,Y 146.016,Z 505.682,A -85,B 0,C 180,E1 -24816.984,E2 -24816.984} C_VEL
LIN {X 0,Y 143.376,Z 503.593,A -85,B 0,C 180,E1 -24819.937,E2 -24819.937} C_VEL
LIN {X 0,Y 141.411,Z 500.196,A -85,B 0,C 180,E1 -24822.842,E2 -24822.842} C_VEL
LIN {X 0,Y 138.324,Z 497.953,A -85,B 0,C 180,E1 -24828.279,E2 -24828.279} C_VEL
LIN {X 0,Y 136.692,Z 494.752,A -85,B 0,C 180,E1 -24834.473,E2 -24834.473} C_VEL
LIN {X 0,Y 137.106,Z 493.986,A -85,B 0,C 180,E1 -24840.004,E2 -24840.004} C_VEL
LIN {X 0,Y 136.691,Z 494.778,A -85,B 0,C 180,E1 -24845.167,E2 -24845.167} C_VEL
LIN {X 0,Y 139.961,Z 499.405,A -85,B 0,C 180,E1 -24854.545,E2 -24854.545} C_VEL
LIN {X 0,Y 141.656,Z 500.47,A -85,B 0,C 180,E1 -24857.137,E2 -24857.137} C_VEL
LIN {X 0,Y 143.397,Z 503.582,A -85,B 0,C 180,E1 -24859.695,E2 -24859.695} C_VEL
LIN {X 0,Y 146.177,Z 505.96,A -85,B 0,C 180,E1 -24862.812,E2 -24862.812} C_VEL
LIN {X 0,Y 148.235,Z 509.19,A -85,B 0,C 180,E1 -24864.981,E2 -24864.981} C_VEL
LIN {X 0,Y 150.388,Z 511.318,A -85,B 0,C 180,E1 -24866.892,E2 -24866.892} C_VEL
LIN {X 0,Y 153.133,Z 515.068,A -85,B 0,C 180,E1 -24869.19,E2 -24869.19} C_VEL
LIN {X 0,Y 154.284,Z 516.564,A -85,B 0,C 180,E1 -24870.075,E2 -24870.075} C_VEL
LIN {X 0,Y 157.379,Z 520.873,A -85,B 0,C 180,E1 -24872.314,E2 -24872.314} C_VEL
LIN {X 0,Y 159.869,Z 524.84,A -85,B 0,C 180,E1 -24874,E2 -24874} C_VEL
LIN {X 0,Y 163.836,Z 532.297,A -85,B 0,C 180,E1 -24876.53,E2 -24876.53} C_VEL
LIN {X 0,Y 169.74,Z 544.933,A -85,B 0,C 180,E1 -24879.943,E2 -24879.943} C_VEL
LIN {X 0,Y 174.629,Z 557.896,A -85,B 0,C 180,E1 -24882.585,E2 -24882.585} C_VEL
LIN {X 0,Y 175.25,Z 560.976,A -85,B 0,C 180,E1 -24882.984,E2 -24882.984} C_VEL
LIN {X 0,Y 172.693,Z 597.042,A -85,B 0,C 180,E1 -24884.326,E2 -24884.326} C_VEL
LIN {X 0,Y 171.205,Z 607.916,A -85,B 0,C 180,E1 -24884.973,E2 -24884.973} C_VEL
LIN {X 0,Y 169.022,Z 618.654,A -85,B 0,C 180,E1 -24885.856,E2 -24885.856} C_VEL
LIN {X 0,Y 165.816,Z 631.101,A -85,B 0,C 180,E1 -24887.302,E2 -24887.302} C_VEL
LIN {X 0,Y 161.606,Z 643.359,A -85,B 0,C 180,E1 -24889.283,E2 -24889.283} C_VEL
LIN {X 0,Y 158.227,Z 652.083,A -85,B 0,C 180,E1 -24891.142,E2 -24891.142} C_VEL
LIN {X 0,Y 154.947,Z 659.499,A -85,B 0,C 180,E1 -24893.06,E2 -24893.06} C_VEL
LIN {X 0,Y 150.637,Z 668.29,A -85,B 0,C 180,E1 -24895.954,E2 -24895.954} C_VEL
LIN {X 0,Y 147.59,Z 674.281,A -85,B 0,C 180,E1 -24898.413,E2 -24898.413} C_VEL
LIN {X 0,Y 144.221,Z 680.594,A -85,B 0,C 180,E1 -24901.633,E2 -24901.633} C_VEL
LIN {X 0,Y 141.146,Z 685.866,A -85,B 0,C 180,E1 -24904.961,E2 -24904.961} C_VEL
LIN {X 0,Y 138.132,Z 690.961,A -85,B 0,C 180,E1 -24909.136,E2 -24909.136} C_VEL
LIN {X 0,Y 135.875,Z 694.929,A -85,B 0,C 180,E1 -24913.472,E2 -24913.472} C_VEL
LIN {X 0,Y 134.44,Z 697.873,A -85,B 0,C 180,E1 -24917.93,E2 -24917.93} C_VEL
LIN {X 0,Y 133.815,Z 699.379,A -85,B 0,C 180,E1 -24920.935,E2 -24920.935} C_VEL
LIN {X 0,Y 133.405,Z 700.917,A -85,B 0,C 180,E1 -24926.98,E2 -24926.98} C_VEL
LIN {X 0,Y 133.504,Z 701.201,A -85,B 0,C 180,E1 -24930,E2 -24930} C_VEL
LIN {X 0,Y 133.471,Z 700.314,A -85,B 0,C 180,E1 -24936.045,E2 -24936.045} C_VEL
LIN {X 0,Y 133.822,Z 699.379,A -85,B 0,C 180,E1 -24939.065,E2 -24939.065} C_VEL
LIN {X 0,Y 135.334,Z 696.022,A -85,B 0,C 180,E1 -24945.049,E2 -24945.049} C_VEL
LIN {X 0,Y 137.284,Z 692.389,A -85,B 0,C 180,E1 -24949.436,E2 -24949.436} C_VEL
LIN {X 0,Y 140.064,Z 687.657,A -85,B 0,C 180,E1 -24953.667,E2 -24953.667} C_VEL
LIN {X 0,Y 143.595,Z 681.687,A -85,B 0,C 180,E1 -24957.707,E2 -24957.707} C_VEL
LIN {X 0,Y 146.891,Z 675.595,A -85,B 0,C 180,E1 -24960.952,E2 -24960.952} C_VEL
LIN {X 0,Y 149.868,Z 669.852,A -85,B 0,C 180,E1 -24963.436,E2 -24963.436} C_VEL
LIN {X 0,Y 153.2,Z 663.199,A -85,B 0,C 180,E1 -24965.796,E2 -24965.796} C_VEL
LIN {X 0,Y 156.765,Z 655.375,A -85,B 0,C 180,E1 -24968.056,E2 -24968.056} C_VEL
LIN {X 0,Y 160.169,Z 647.298,A -85,B 0,C 180,E1 -24969.92,E2 -24969.92} C_VEL
LIN {X 0,Y 163.679,Z 637.541,A -85,B 0,C 180,E1 -24971.723,E2 -24971.723} C_VEL
LIN {X 0,Y 166.28,Z 629.154,A -85,B 0,C 180,E1 -24972.964,E2 -24972.964} C_VEL
LIN {X 0,Y 168.979,Z 618.652,A -85,B 0,C 180,E1 -24974.158,E2 -24974.158} C_VEL
LIN {X 0,Y 171.189,Z 607.911,A -85,B 0,C 180,E1 -24975.033,E2 -24975.033} C_VEL
LIN {X 0,Y 171.292,Z 607.37,A -85,B 0,C 180,E1 -24975.063,E2 -24975.063} C_VEL
LIN {X 0,Y 171.908,Z 601.667,A -85,B 0,C 180,E1 -24975.542,E2 -24975.542} C_VEL
LIN {X 0,Y 170.846,Z 592.409,A -85,B 0,C 180,E1 -24976.67,E2 -24976.67} C_VEL
LIN {X 0,Y 169.47,Z 583.087,A -85,B 0,C 180,E1 -24977.771,E2 -24977.771} C_VEL
LIN {X 0,Y 169.352,Z 577.267,A -85,B 0,C 180,E1 -24978.165,E2 -24978.165} C_VEL
LIN {X 0,Y 170.352,Z 561.848,A -85,B 0,C 180,E1 -24978.747,E2 -24978.747} C_VEL
LIN {X 0,Y 165.618,Z 548.901,A -85,B 0,C 180,E1 -24981.508,E2 -24981.508} C_VEL
LIN {X 0,Y 159.847,Z 536.137,A -85,B 0,C 180,E1 -24985.136,E2 -24985.136} C_VEL
LIN {X 0,Y 155.569,Z 528.111,A -85,B 0,C 180,E1 -24988.126,E2 -24988.126} C_VEL
LIN {X 0,Y 153.223,Z 524.679,A -85,B 0,C 180,E1 -24989.865,E2 -24989.865} C_VEL
LIN {X 0,Y 150.751,Z 521.202,A -85,B 0,C 180,E1 -24991.852,E2 -24991.852} C_VEL
LIN {X 0,Y 147.651,Z 516.988,A -85,B 0,C 180,E1 -24994.63,E2 -24994.63} C_VEL
LIN {X 0,Y 144.852,Z 513.53,A -85,B 0,C 180,E1 -24997.484,E2 -24997.484} C_VEL
LIN {X 0,Y 143.938,Z 512.165,A -85,B 0,C 180,E1 -24998.55,E2 -24998.55} C_VEL
LIN {X 0,Y 141.276,Z 509.463,A -85,B 0,C 180,E1 -25001.881,E2 -25001.881} C_VEL
LIN {X 0,Y 140.006,Z 506.952,A -85,B 0,C 180,E1 -25003.969,E2 -25003.969} C_VEL
LIN {X 0,Y 137.39,Z 505.055,A -85,B 0,C 180,E1 -25008.759,E2 -25008.759} C_VEL
LIN {X 0,Y 135.532,Z 501.62,A -85,B 0,C 180,E1 -25015.534,E2 -25015.534} C_VEL
LIN {X 0,Y 135.181,Z 500.835,A -85,B 0,C 180,E1 -25019.995,E2 -25019.995} C_VEL
LIN {X 0,Y 135.585,Z 501.744,A -85,B 0,C 180,E1 -25025.2,E2 -25025.2} C_VEL
LIN {X 0,Y 138.594,Z 506.206,A -85,B 0,C 180,E1 -25034.12,E2 -25034.12} C_VEL
LIN {X 0,Y 140.149,Z 507.181,A -85,B 0,C 180,E1 -25036.66,E2 -25036.66} C_VEL
LIN {X 0,Y 141.993,Z 510.459,A -85,B 0,C 180,E1 -25039.513,E2 -25039.513} C_VEL
LIN {X 0,Y 144.369,Z 512.624,A -85,B 0,C 180,E1 -25042.325,E2 -25042.325} C_VEL
LIN {X 0,Y 146.953,Z 516.35,A -85,B 0,C 180,E1 -25045.111,E2 -25045.111} C_VEL
LIN {X 0,Y 148.299,Z 517.778,A -85,B 0,C 180,E1 -25046.362,E2 -25046.362} C_VEL
LIN {X 0,Y 151.133,Z 521.579,A -85,B 0,C 180,E1 -25048.841,E2 -25048.841} C_VEL
LIN {X 0,Y 155.262,Z 527.671,A -85,B 0,C 180,E1 -25052.044,E2 -25052.044} C_VEL
LIN {X 0,Y 159.627,Z 534.305,A -85,B 0,C 180,E1 -25054.999,E2 -25054.999} C_VEL
LIN {X 0,Y 165.413,Z 544.185,A -85,B 0,C 180,E1 -25058.469,E2 -25058.469} C_VEL
LIN {X 0,Y 171.102,Z 555.482,A -85,B 0,C 180,E1 -25061.531,E2 -25061.531} C_VEL
LIN {X 0,Y 176.04,Z 567.441,A -85,B 0,C 180,E1 -25064.021,E2 -25064.021} C_VEL
LIN {X 0,Y 182.739,Z 583.885,A -85,B 0,C 180,E1 -25067.043,E2 -25067.043} C_VEL
LIN {X 0,Y 188.862,Z 596.671,A -85,B 0,C 180,E1 -25069.71,E2 -25069.71} C_VEL
LIN {X 0,Y 193.904,Z 606.078,A -85,B 0,C 180,E1 -25071.964,E2 -25071.964} C_VEL
LIN {X 0,Y 200.129,Z 616.312,A -85,B 0,C 180,E1 -25074.728,E2 -25074.728} C_VEL
LIN {X 0,Y 206.15,Z 624.795,A -85,B 0,C 180,E1 -25077.259,E2 -25077.259} C_VEL
LIN {X 0,Y 213.221,Z 633.443,A -85,B 0,C 180,E1 -25080.067,E2 -25080.067} C_VEL
LIN {X 0,Y 222.556,Z 642.913,A -85,B 0,C 180,E1 -25083.435,E2 -25083.435} C_VEL
LIN {X 0,Y 234.021,Z 652.034,A -85,B 0,C 180,E1 -25087.02,E2 -25087.02} C_VEL
LIN {X 0,Y 246.253,Z 659.85,A -85,B 0,C 180,E1 -25090.349,E2 -25090.349} C_VEL
LIN {X 0,Y 259.102,Z 666.948,A -85,B 0,C 180,E1 -25093.558,E2 -25093.558} C_VEL
LIN {X 0,Y 268.177,Z 671.766,A -85,B 0,C 180,E1 -25095.834,E2 -25095.834} C_VEL
LIN {X 0,Y 273.735,Z 674.762,A -85,B 0,C 180,E1 -25097.311,E2 -25097.311} C_VEL
LIN {X 0,Y 279.291,Z 677.838,A -85,B 0,C 180,E1 -25098.912,E2 -25098.912} C_VEL
LIN {X 0,Y 284.866,Z 680.944,A -85,B 0,C 180,E1 -25100.68,E2 -25100.68} C_VEL
LIN {X 0,Y 288.725,Z 683.474,A -85,B 0,C 180,E1 -25102.307,E2 -25102.307} C_VEL
LIN {X 0,Y 290.308,Z 684.509,A -85,B 0,C 180,E1 -25103.048,E2 -25103.048} C_VEL
LIN {X 0,Y 293.087,Z 686.099,A -85,B 0,C 180,E1 -25104.496,E2 -25104.496} C_VEL
LIN {X 0,Y 295.818,Z 687.491,A -85,B 0,C 180,E1 -25106.18,E2 -25106.18} C_VEL
LIN {X 0,Y 297.161,Z 688.118,A -85,B 0,C 180,E1 -25107.289,E2 -25107.289} C_VEL
LIN {X 0,Y 298.281,Z 688.537,A -85,B 0,C 180,E1 -25108.65,E2 -25108.65} C_VEL
LIN {X 0,Y 298.847,Z 688.638,A -85,B 0,C 180,E1 -25110,E2 -25110} C_VEL
LIN {X 0,Y 298.288,Z 688.543,A -85,B 0,C 180,E1 -25111.35,E2 -25111.35} C_VEL
LIN {X 0,Y 297.174,Z 688.133,A -85,B 0,C 180,E1 -25112.711,E2 -25112.711} C_VEL
LIN {X 0,Y 295.373,Z 687.328,A -85,B 0,C 180,E1 -25114.093,E2 -25114.093} C_VEL
LIN {X 0,Y 293.035,Z 686.11,A -85,B 0,C 180,E1 -25115.505,E2 -25115.505} C_VEL
LIN {X 0,Y 290.268,Z 684.511,A -85,B 0,C 180,E1 -25116.953,E2 -25116.953} C_VEL
LIN {X 0,Y 286.991,Z 682.36,A -85,B 0,C 180,E1 -25118.449,E2 -25118.449} C_VEL
LIN {X 0,Y 282.789,Z 679.742,A -85,B 0,C 180,E1 -25120.018,E2 -25120.018} C_VEL
LIN {X 0,Y 277.211,Z 676.691,A -85,B 0,C 180,E1 -25121.702,E2 -25121.702} C_VEL
LIN {X 0,Y 270.741,Z 673.112,A -85,B 0,C 180,E1 -25123.51,E2 -25123.51} C_VEL
LIN {X 0,Y 261.122,Z 668.044,A -85,B 0,C 180,E1 -25125.946,E2 -25125.946} C_VEL
LIN {X 0,Y 248.935,Z 661.429,A -85,B 0,C 180,E1 -25128.964,E2 -25128.964} C_VEL
LIN {X 0,Y 235.764,Z 653.258,A -85,B 0,C 180,E1 -25132.477,E2 -25132.477} C_VEL
LIN {X 0,Y 224.103,Z 644.273,A -85,B 0,C 180,E1 -25136.043,E2 -25136.043} C_VEL
LIN {X 0,Y 215.152,Z 635.524,A -85,B 0,C 180,E1 -25139.2,E2 -25139.2} C_VEL
LIN {X 0,Y 206.132,Z 624.865,A -85,B 0,C 180,E1 -25142.732,E2 -25142.732} C_VEL
LIN {X 0,Y 198.216,Z 613.333,A -85,B 0,C 180,E1 -25146.126,E2 -25146.126} C_VEL
LIN {X 0,Y 191.557,Z 601.796,A -85,B 0,C 180,E1 -25149.092,E2 -25149.092} C_VEL
LIN {X 0,Y 185.784,Z 590.339,A -85,B 0,C 180,E1 -25151.664,E2 -25151.664} C_VEL
LIN {X 0,Y 179.785,Z 577.14,A -85,B 0,C 180,E1 -25154.215,E2 -25154.215} C_VEL
LIN {X 0,Y 173.121,Z 560.167,A -85,B 0,C 180,E1 -25157.432,E2 -25157.432} C_VEL
LIN {X 0,Y 168.745,Z 550.625,A -85,B 0,C 180,E1 -25159.7,E2 -25159.7} C_VEL
LIN {X 0,Y 163.845,Z 541.445,A -85,B 0,C 180,E1 -25162.424,E2 -25162.424} C_VEL
LIN {X 0,Y 158.884,Z 533.117,A -85,B 0,C 180,E1 -25165.482,E2 -25165.482} C_VEL
LIN {X 0,Y 153.696,Z 525.299,A -85,B 0,C 180,E1 -25169.121,E2 -25169.121} C_VEL
LIN {X 0,Y 150.754,Z 521.206,A -85,B 0,C 180,E1 -25171.46,E2 -25171.46} C_VEL
LIN {X 0,Y 147.649,Z 516.994,A -85,B 0,C 180,E1 -25174.243,E2 -25174.243} C_VEL
LIN {X 0,Y 144.939,Z 513.702,A -85,B 0,C 180,E1 -25176.992,E2 -25176.992} C_VEL
LIN {X 0,Y 144.048,Z 512.246,A -85,B 0,C 180,E1 -25178.041,E2 -25178.041} C_VEL
LIN {X 0,Y 141.561,Z 509.867,A -85,B 0,C 180,E1 -25181.084,E2 -25181.084} C_VEL
LIN {X 0,Y 139.991,Z 506.943,A -85,B 0,C 180,E1 -25183.602,E2 -25183.602} C_VEL
LIN {X 0,Y 137.231,Z 504.885,A -85,B 0,C 180,E1 -25188.747,E2 -25188.747} C_VEL
LIN {X 0,Y 135.529,Z 501.599,A -85,B 0,C 180,E1 -25195.171,E2 -25195.171} C_VEL
LIN {X 0,Y 135.182,Z 500.83,A -85,B 0,C 180,E1 -25200.005,E2 -25200.005} C_VEL
LIN {X 0,Y 135.653,Z 501.891,A -85,B 0,C 180,E1 -25205.206,E2 -25205.206} C_VEL
LIN {X 0,Y 138.706,Z 506.272,A -85,B 0,C 180,E1 -25213.931,E2 -25213.931} C_VEL
LIN {X 0,Y 140.16,Z 507.219,A -85,B 0,C 180,E1 -25216.294,E2 -25216.294} C_VEL
LIN {X 0,Y 142.014,Z 510.43,A -85,B 0,C 180,E1 -25219.143,E2 -25219.143} C_VEL
LIN {X 0,Y 144.439,Z 512.764,A -85,B 0,C 180,E1 -25222.023,E2 -25222.023} C_VEL
LIN {X 0,Y 146.972,Z 516.36,A -85,B 0,C 180,E1 -25224.739,E2 -25224.739} C_VEL
LIN {X 0,Y 148.381,Z 517.897,A -85,B 0,C 180,E1 -25226.05,E2 -25226.05} C_VEL
LIN {X 0,Y 151.975,Z 522.849,A -85,B 0,C 180,E1 -25229.149,E2 -25229.149} C_VEL
LIN {X 0,Y 154.969,Z 527.202,A -85,B 0,C 180,E1 -25231.44,E2 -25231.44} C_VEL
LIN {X 0,Y 156.764,Z 530.241,A -85,B 0,C 180,E1 -25232.741,E2 -25232.741} C_VEL
LIN {X 0,Y 160.265,Z 537.014,A -85,B 0,C 180,E1 -25235.143,E2 -25235.143} C_VEL
LIN {X 0,Y 165.962,Z 549.731,A -85,B 0,C 180,E1 -25238.696,E2 -25238.696} C_VEL
LIN {X 0,Y 170.411,Z 562.134,A -85,B 0,C 180,E1 -25241.294,E2 -25241.294} C_VEL
LIN {X 0,Y 167.838,Z 596.566,A -85,B 0,C 180,E1 -25242.577,E2 -25242.577} C_VEL
LIN {X 0,Y 166.305,Z 607.571,A -85,B 0,C 180,E1 -25243.238,E2 -25243.238} C_VEL
LIN {X 0,Y 164.017,Z 618.458,A -85,B 0,C 180,E1 -25244.134,E2 -25244.134} C_VEL
LIN {X 0,Y 160.664,Z 630.904,A -85,B 0,C 180,E1 -25245.582,E2 -25245.582} C_VEL
LIN {X 0,Y 156.299,Z 643.163,A -85,B 0,C 180,E1 -25247.587,E2 -25247.587} C_VEL
LIN {X 0,Y 152.749,Z 651.887,A -85,B 0,C 180,E1 -25249.467,E2 -25249.467} C_VEL
LIN {X 0,Y 149.313,Z 659.303,A -85,B 0,C 180,E1 -25251.416,E2 -25251.416} C_VEL
LIN {X 0,Y 144.803,Z 668.094,A -85,B 0,C 180,E1 -25254.38,E2 -25254.38} C_VEL
LIN {X 0,Y 141.551,Z 674.083,A -85,B 0,C 180,E1 -25256.897,E2 -25256.897} C_VEL
LIN {X 0,Y 138.104,Z 680.194,A -85,B 0,C 180,E1 -25260.097,E2 -25260.097} C_VEL
LIN {X 0,Y 134.734,Z 685.67,A -85,B 0,C 180,E1 -25263.681,E2 -25263.681} C_VEL
LIN {X 0,Y 131.497,Z 690.764,A -85,B 0,C 180,E1 -25268.03,E2 -25268.03} C_VEL
LIN {X 0,Y 129.054,Z 694.732,A -85,B 0,C 180,E1 -25272.572,E2 -25272.572} C_VEL
LIN {X 0,Y 127.47,Z 697.676,A -85,B 0,C 180,E1 -25277.259,E2 -25277.259} C_VEL
LIN {X 0,Y 126.788,Z 699.182,A -85,B 0,C 180,E1 -25280.428,E2 -25280.428} C_VEL
LIN {X 0,Y 126.311,Z 700.72,A -85,B 0,C 180,E1 -25286.81,E2 -25286.81} C_VEL
LIN {X 0,Y 126.428,Z 701.006,A -85,B 0,C 180,E1 -25290,E2 -25290} C_VEL
LIN {X 0,Y 126.414,Z 700.117,A -85,B 0,C 180,E1 -25296.384,E2 -25296.384} C_VEL
LIN {X 0,Y 126.793,Z 699.183,A -85,B 0,C 180,E1 -25299.572,E2 -25299.572} C_VEL
LIN {X 0,Y 128.452,Z 695.824,A -85,B 0,C 180,E1 -25305.876,E2 -25305.876} C_VEL
LIN {X 0,Y 130.583,Z 692.192,A -85,B 0,C 180,E1 -25310.477,E2 -25310.477} C_VEL
LIN {X 0,Y 133.552,Z 687.459,A -85,B 0,C 180,E1 -25314.897,E2 -25314.897} C_VEL
LIN {X 0,Y 137.318,Z 681.49,A -85,B 0,C 180,E1 -25319.092,E2 -25319.092} C_VEL
LIN {X 0,Y 140.818,Z 675.397,A -85,B 0,C 180,E1 -25322.446,E2 -25322.446} C_VEL
LIN {X 0,Y 143.965,Z 669.654,A -85,B 0,C 180,E1 -25325.002,E2 -25325.002} C_VEL
LIN {X 0,Y 147.473,Z 663.002,A -85,B 0,C 180,E1 -25327.417,E2 -25327.417} C_VEL
LIN {X 0,Y 151.239,Z 655.179,A -85,B 0,C 180,E1 -25329.714,E2 -25329.714} C_VEL
LIN {X 0,Y 154.774,Z 647.101,A -85,B 0,C 180,E1 -25331.612,E2 -25331.612} C_VEL
LIN {X 0,Y 158.452,Z 637.345,A -85,B 0,C 180,E1 -25333.431,E2 -25333.431} C_VEL
LIN {X 0,Y 161.156,Z 628.958,A -85,B 0,C 180,E1 -25334.684,E2 -25334.684} C_VEL
LIN {X 0,Y 163.963,Z 618.456,A -85,B 0,C 180,E1 -25335.886,E2 -25335.886} C_VEL
LIN {X 0,Y 166.148,Z 608.296,A -85,B 0,C 180,E1 -25336.726,E2 -25336.726} C_VEL
LIN {X 0,Y 167.747,Z 597.622,A -85,B 0,C 180,E1 -25337.357,E2 -25337.357} C_VEL
LIN {X 0,Y 169.352,Z 577.267,A -85,B 0,C 180,E1 -25338.165,E2 -25338.165} C_VEL
LIN {X 0,Y 169.13,Z 573.477,A -85,B 0,C 180,E1 -25338.485,E2 -25338.485} C_VEL
LIN {X 0,Y 168.234,Z 569.988,A -85,B 0,C 180,E1 -25339.05,E2 -25339.05} C_VEL
LIN {X 0,Y 163.901,Z 559.182,A -85,B 0,C 180,E1 -25341.552,E2 -25341.552} C_VEL
LIN {X 0,Y 161.021,Z 551.504,A -85,B 0,C 180,E1 -25343.409,E2 -25343.409} C_VEL
LIN {X 0,Y 156.189,Z 540.501,A -85,B 0,C 180,E1 -25346.739,E2 -25346.739} C_VEL
LIN {X 0,Y 152.598,Z 533.52,A -85,B 0,C 180,E1 -25349.462,E2 -25349.462} C_VEL
LIN {X 0,Y 148.824,Z 527.773,A -85,B 0,C 180,E1 -25352.581,E2 -25352.581} C_VEL
LIN {X 0,Y 145.473,Z 523.205,A -85,B 0,C 180,E1 -25355.75,E2 -25355.75} C_VEL
LIN {X 0,Y 142.782,Z 519.577,A -85,B 0,C 180,E1 -25358.729,E2 -25358.729} C_VEL
LIN {X 0,Y 141.966,Z 518.607,A -85,B 0,C 180,E1 -25359.72,E2 -25359.72} C_VEL
LIN {X 0,Y 139.343,Z 515.377,A -85,B 0,C 180,E1 -25363.392,E2 -25363.392} C_VEL
LIN {X 0,Y 138.6,Z 513.773,A -85,B 0,C 180,E1 -25364.745,E2 -25364.745} C_VEL
LIN {X 0,Y 136.169,Z 511.794,A -85,B 0,C 180,E1 -25369.571,E2 -25369.571} C_VEL
LIN {X 0,Y 134.555,Z 508.517,A -85,B 0,C 180,E1 -25376.252,E2 -25376.252} C_VEL
LIN {X 0,Y 134.317,Z 507.872,A -85,B 0,C 180,E1 -25379.995,E2 -25379.995} C_VEL
LIN {X 0,Y 134.697,Z 508.854,A -85,B 0,C 180,E1 -25385.14,E2 -25385.14} C_VEL
LIN {X 0,Y 137.57,Z 513.21,A -85,B 0,C 180,E1 -25393.886,E2 -25393.886} C_VEL
LIN {X 0,Y 138.732,Z 514.037,A -85,B 0,C 180,E1 -25395.89,E2 -25395.89} C_VEL
LIN {X 0,Y 140.626,Z 517.308,A -85,B 0,C 180,E1 -25398.951,E2 -25398.951} C_VEL
LIN {X 0,Y 142.718,Z 519.44,A -85,B 0,C 180,E1 -25401.575,E2 -25401.575} C_VEL
LIN {X 0,Y 145.295,Z 523.025,A -85,B 0,C 180,E1 -25404.462,E2 -25404.462} C_VEL
LIN {X 0,Y 146.522,Z 524.677,A -85,B 0,C 180,E1 -25405.691,E2 -25405.691} C_VEL
LIN {X 0,Y 149.693,Z 529.112,A -85,B 0,C 180,E1 -25408.569,E2 -25408.569} C_VEL
LIN {X 0,Y 154.196,Z 535.917,A -85,B 0,C 180,E1 -25412.119,E2 -25412.119} C_VEL
LIN {X 0,Y 159.869,Z 545.51,A -85,B 0,C 180,E1 -25415.976,E2 -25415.976} C_VEL
LIN {X 0,Y 164.684,Z 554.799,A -85,B 0,C 180,E1 -25418.878,E2 -25418.878} C_VEL
LIN {X 0,Y 169.026,Z 564.52,A -85,B 0,C 180,E1 -25421.3,E2 -25421.3} C_VEL
LIN {X 0,Y 178.023,Z 587.756,A -85,B 0,C 180,E1 -25425.884,E2 -25425.884} C_VEL
LIN {X 0,Y 182.444,Z 597.659,A -85,B 0,C 180,E1 -25428.063,E2 -25428.063} C_VEL
LIN {X 0,Y 187.195,Z 607.431,A -85,B 0,C 180,E1 -25430.497,E2 -25430.497} C_VEL
LIN {X 0,Y 191.736,Z 615.797,A -85,B 0,C 180,E1 -25432.8,E2 -25432.8} C_VEL
LIN {X 0,Y 198.75,Z 626.665,A -85,B 0,C 180,E1 -25436.193,E2 -25436.193} C_VEL
LIN {X 0,Y 206.06,Z 636.095,A -85,B 0,C 180,E1 -25439.441,E2 -25439.441} C_VEL
LIN {X 0,Y 214.086,Z 644.573,A -85,B 0,C 180,E1 -25442.64,E2 -25442.64} C_VEL
LIN {X 0,Y 223.326,Z 652.385,A -85,B 0,C 180,E1 -25445.862,E2 -25445.862} C_VEL
LIN {X 0,Y 236.055,Z 660.879,A -85,B 0,C 180,E1 -25449.682,E2 -25449.682} C_VEL
LIN {X 0,Y 249.546,Z 668.199,A -85,B 0,C 180,E1 -25453.234,E2 -25453.234} C_VEL
LIN {X 0,Y 260.67,Z 673.671,A -85,B 0,C 180,E1 -25456.061,E2 -25456.061} C_VEL
LIN {X 0,Y 269.174,Z 677.843,A -85,B 0,C 180,E1 -25458.363,E2 -25458.363} C_VEL
LIN {X 0,Y 275.918,Z 681.191,A -85,B 0,C 180,E1 -25460.373,E2 -25460.373} C_VEL
LIN {X 0,Y 278.677,Z 682.593,A -85,B 0,C 180,E1 -25461.297,E2 -25461.297} C_VEL
LIN {X 0,Y 283.082,Z 685.19,A -85,B 0,C 180,E1 -25463.225,E2 -25463.225} C_VEL
LIN {X 0,Y 285.257,Z 686.45,A -85,B 0,C 180,E1 -25464.344,E2 -25464.344} C_VEL
LIN {X 0,Y 288.718,Z 688.197,A -85,B 0,C 180,E1 -25466.354,E2 -25466.354} C_VEL
LIN {X 0,Y 289.829,Z 688.68,A -85,B 0,C 180,E1 -25467.22,E2 -25467.22} C_VEL
LIN {X 0,Y 291.088,Z 689.186,A -85,B 0,C 180,E1 -25468.617,E2 -25468.617} C_VEL
LIN {X 0,Y 291.765,Z 689.331,A -85,B 0,C 180,E1 -25470,E2 -25470} C_VEL
LIN {X 0,Y 291.096,Z 689.189,A -85,B 0,C 180,E1 -25471.383,E2 -25471.383} C_VEL
LIN {X 0,Y 289.83,Z 688.681,A -85,B 0,C 180,E1 -25472.78,E2 -25472.78} C_VEL
LIN {X 0,Y 287.776,Z 687.766,A -85,B 0,C 180,E1 -25474.202,E2 -25474.202} C_VEL
LIN {X 0,Y 285.214,Z 686.452,A -85,B 0,C 180,E1 -25475.656,E2 -25475.656} C_VEL
LIN {X 0,Y 282.258,Z 684.744,A -85,B 0,C 180,E1 -25477.152,E2 -25477.152} C_VEL
LIN {X 0,Y 277.552,Z 682.024,A -85,B 0,C 180,E1 -25479.076,E2 -25479.076} C_VEL
LIN {X 0,Y 271.906,Z 679.214,A -85,B 0,C 180,E1 -25480.845,E2 -25480.845} C_VEL
LIN {X 0,Y 263.488,Z 674.99,A -85,B 0,C 180,E1 -25483.217,E2 -25483.217} C_VEL
LIN {X 0,Y 251.781,Z 669.285,A -85,B 0,C 180,E1 -25486.208,E2 -25486.208} C_VEL
LIN {X 0,Y 238.724,Z 662.397,A -85,B 0,C 180,E1 -25489.607,E2 -25489.607} C_VEL
LIN {X 0,Y 225.806,Z 654.194,A -85,B 0,C 180,E1 -25493.35,E2 -25493.35} C_VEL
LIN {X 0,Y 216.142,Z 646.469,A -85,B 0,C 180,E1 -25496.607,E2 -25496.607} C_VEL
LIN {X 0,Y 207.157,Z 637.288,A -85,B 0,C 180,E1 -25500.114,E2 -25500.114} C_VEL
LIN {X 0,Y 199.76,Z 628.101,A -85,B 0,C 180,E1 -25503.331,E2 -25503.331} C_VEL
LIN {X 0,Y 193.74,Z 619.12,A -85,B 0,C 180,E1 -25506.189,E2 -25506.189} C_VEL
LIN {X 0,Y 188.898,Z 610.688,A -85,B 0,C 180,E1 -25508.626,E2 -25508.626} C_VEL
LIN {X 0,Y 183.757,Z 600.509,A -85,B 0,C 180,E1 -25511.262,E2 -25511.262} C_VEL
LIN {X 0,Y 178.689,Z 589.226,A -85,B 0,C 180,E1 -25513.829,E2 -25513.829} C_VEL
LIN {X 0,Y 172.385,Z 573.378,A -85,B 0,C 180,E1 -25516.902,E2 -25516.902} C_VEL
LIN {X 0,Y 167.939,Z 561.913,A -85,B 0,C 180,E1 -25519.294,E2 -25519.294} C_VEL
LIN {X 0,Y 162.996,Z 551.391,A -85,B 0,C 180,E1 -25522.109,E2 -25522.109} C_VEL
LIN {X 0,Y 157.653,Z 541.613,A -85,B 0,C 180,E1 -25525.465,E2 -25525.465} C_VEL
LIN {X 0,Y 153.185,Z 534.415,A -85,B 0,C 180,E1 -25528.626,E2 -25528.626} C_VEL
LIN {X 0,Y 150.14,Z 529.831,A -85,B 0,C 180,E1 -25531.046,E2 -25531.046} C_VEL
LIN {X 0,Y 148.299,Z 527.159,A -85,B 0,C 180,E1 -25532.646,E2 -25532.646} C_VEL
LIN {X 0,Y 145.617,Z 523.389,A -85,B 0,C 180,E1 -25535.215,E2 -25535.215} C_VEL
LIN {X 0,Y 142.915,Z 519.826,A -85,B 0,C 180,E1 -25538.172,E2 -25538.172} C_VEL
LIN {X 0,Y 142.024,Z 518.654,A -85,B 0,C 180,E1 -25539.263,E2 -25539.263} C_VEL
LIN {X 0,Y 139.525,Z 515.727,A -85,B 0,C 180,E1 -25542.697,E2 -25542.697} C_VEL
LIN {X 0,Y 138.483,Z 513.665,A -85,B 0,C 180,E1 -25544.552,E2 -25544.552} C_VEL
LIN {X 0,Y 136.132,Z 511.789,A -85,B 0,C 180,E1 -25549.267,E2 -25549.267} C_VEL
LIN {X 0,Y 134.604,Z 508.6,A -85,B 0,C 180,E1 -25555.513,E2 -25555.513} C_VEL
LIN {X 0,Y 134.317,Z 507.872,A -85,B 0,C 180,E1 -25560.005,E2 -25560.005} C_VEL
LIN {X 0,Y 134.718,Z 508.881,A -85,B 0,C 180,E1 -25564.868,E2 -25564.868} C_VEL
LIN {X 0,Y 137.66,Z 513.265,A -85,B 0,C 180,E1 -25573.662,E2 -25573.662} C_VEL
LIN {X 0,Y 138.746,Z 514.029,A -85,B 0,C 180,E1 -25575.521,E2 -25575.521} C_VEL
LIN {X 0,Y 140.673,Z 517.334,A -85,B 0,C 180,E1 -25578.623,E2 -25578.623} C_VEL
LIN {X 0,Y 142.607,Z 519.247,A -85,B 0,C 180,E1 -25581.046,E2 -25581.046} C_VEL
LIN {X 0,Y 145.472,Z 523.217,A -85,B 0,C 180,E1 -25584.25,E2 -25584.25} C_VEL
LIN {X 0,Y 147.004,Z 525.414,A -85,B 0,C 180,E1 -25585.774,E2 -25585.774} C_VEL
LIN {X 0,Y 149.707,Z 529.143,A -85,B 0,C 180,E1 -25588.194,E2 -25588.194} C_VEL
LIN {X 0,Y 152.695,Z 533.666,A -85,B 0,C 180,E1 -25590.613,E2 -25590.613} C_VEL
LIN {X 0,Y 155.989,Z 540.094,A -85,B 0,C 180,E1 -25593.117,E2 -25593.117} C_VEL
LIN {X 0,Y 160.121,Z 549.385,A -85,B 0,C 180,E1 -25596.001,E2 -25596.001} C_VEL
LIN {X 0,Y 163.38,Z 557.604,A -85,B 0,C 180,E1 -25598.11,E2 -25598.11} C_VEL
LIN {X 0,Y 165.641,Z 564.22,A -85,B 0,C 180,E1 -25599.531,E2 -25599.531} C_VEL
LIN {X 0,Y 163.09,Z 596.575,A -85,B 0,C 180,E1 -25600.748,E2 -25600.748} C_VEL
LIN {X 0,Y 161.471,Z 607.704,A -85,B 0,C 180,E1 -25601.427,E2 -25601.427} C_VEL
LIN {X 0,Y 158.867,Z 619.525,A -85,B 0,C 180,E1 -25602.42,E2 -25602.42} C_VEL
LIN {X 0,Y 155.107,Z 632.383,A -85,B 0,C 180,E1 -25604.004,E2 -25604.004} C_VEL
LIN {X 0,Y 151.139,Z 642.967,A -85,B 0,C 180,E1 -25605.774,E2 -25605.774} C_VEL
LIN {X 0,Y 147.43,Z 651.691,A -85,B 0,C 180,E1 -25607.675,E2 -25607.675} C_VEL
LIN {X 0,Y 143.82,Z 659.106,A -85,B 0,C 180,E1 -25609.649,E2 -25609.649} C_VEL
LIN {X 0,Y 139.09,Z 667.898,A -85,B 0,C 180,E1 -25612.675,E2 -25612.675} C_VEL
LIN {X 0,Y 135.62,Z 673.886,A -85,B 0,C 180,E1 -25615.248,E2 -25615.248} C_VEL
LIN {X 0,Y 131.561,Z 680.595,A -85,B 0,C 180,E1 -25618.935,E2 -25618.935} C_VEL
LIN {X 0,Y 128.4,Z 685.473,A -85,B 0,C 180,E1 -25622.274,E2 -25622.274} C_VEL
LIN {X 0,Y 124.922,Z 690.567,A -85,B 0,C 180,E1 -25626.808,E2 -25626.808} C_VEL
LIN {X 0,Y 122.251,Z 694.535,A -85,B 0,C 180,E1 -25631.568,E2 -25631.568} C_VEL
LIN {X 0,Y 120.529,Z 697.479,A -85,B 0,C 180,E1 -25636.512,E2 -25636.512} C_VEL
LIN {X 0,Y 119.76,Z 698.985,A -85,B 0,C 180,E1 -25639.86,E2 -25639.86} C_VEL
LIN {X 0,Y 119.227,Z 700.524,A -85,B 0,C 180,E1 -25646.621,E2 -25646.621} C_VEL
LIN {X 0,Y 119.339,Z 700.81,A -85,B 0,C 180,E1 -25650,E2 -25650} C_VEL
LIN {X 0,Y 119.337,Z 699.921,A -85,B 0,C 180,E1 -25656.764,E2 -25656.764} C_VEL
LIN {X 0,Y 119.764,Z 698.985,A -85,B 0,C 180,E1 -25660.139,E2 -25660.139} C_VEL
LIN {X 0,Y 121.609,Z 695.627,A -85,B 0,C 180,E1 -25666.795,E2 -25666.795} C_VEL
LIN {X 0,Y 123.013,Z 693.408,A -85,B 0,C 180,E1 -25670.047,E2 -25670.047} C_VEL
LIN {X 0,Y 126.006,Z 689.053,A -85,B 0,C 180,E1 -25674.728,E2 -25674.728} C_VEL
LIN {X 0,Y 129.776,Z 683.479,A -85,B 0,C 180,E1 -25679.169,E2 -25679.169} C_VEL
LIN {X 0,Y 133.306,Z 677.823,A -85,B 0,C 180,E1 -25682.71,E2 -25682.71} C_VEL
LIN {X 0,Y 137.325,Z 671.018,A -85,B 0,C 180,E1 -25686.054,E2 -25686.054} C_VEL
LIN {X 0,Y 141.88,Z 662.805,A -85,B 0,C 180,E1 -25689.165,E2 -25689.165} C_VEL
LIN {X 0,Y 145.85,Z 654.983,A -85,B 0,C 180,E1 -25691.495,E2 -25691.495} C_VEL
LIN {X 0,Y 149.541,Z 646.905,A -85,B 0,C 180,E1 -25693.419,E2 -25693.419} C_VEL
LIN {X 0,Y 153.378,Z 637.149,A -85,B 0,C 180,E1 -25695.253,E2 -25695.253} C_VEL
LIN {X 0,Y 156.192,Z 628.762,A -85,B 0,C 180,E1 -25696.515,E2 -25696.515} C_VEL
LIN {X 0,Y 159.106,Z 618.26,A -85,B 0,C 180,E1 -25697.72,E2 -25697.72} C_VEL
LIN {X 0,Y 161.342,Z 608.22,A -85,B 0,C 180,E1 -25698.554,E2 -25698.554} C_VEL
LIN {X 0,Y 163.025,Z 597.326,A -85,B 0,C 180,E1 -25699.2,E2 -25699.2} C_VEL
LIN {X 0,Y 164.904,Z 574.438,A -85,B 0,C 180,E1 -25700.097,E2 -25700.097} C_VEL
LIN {X 0,Y 165.64,Z 564.23,A -85,B 0,C 180,E1 -25700.469,E2 -25700.469} C_VEL
LIN {X 0,Y 163.901,Z 559.182,A -85,B 0,C 180,E1 -25701.552,E2 -25701.552} C_VEL
LIN {X 0,Y 162.69,Z 556.14,A -85,B 0,C 180,E1 -25702.302,E2 -25702.302} C_VEL
LIN {X 0,Y 160.245,Z 552.492,A -85,B 0,C 180,E1 -25703.708,E2 -25703.708} C_VEL
LIN {X 0,Y 153.019,Z 544.851,A -85,B 0,C 180,E1 -25708.2,E2 -25708.2} C_VEL
LIN {X 0,Y 150.929,Z 541.166,A -85,B 0,C 180,E1 -25709.832,E2 -25709.832} C_VEL
LIN {X 0,Y 148.361,Z 536.76,A -85,B 0,C 180,E1 -25712.009,E2 -25712.009} C_VEL
LIN {X 0,Y 145.787,Z 532.954,A -85,B 0,C 180,E1 -25714.378,E2 -25714.378} C_VEL
LIN {X 0,Y 143.506,Z 529.602,A -85,B 0,C 180,E1 -25716.739,E2 -25716.739} C_VEL
LIN {X 0,Y 140.436,Z 525.318,A -85,B 0,C 180,E1 -25720.443,E2 -25720.443} C_VEL
LIN {X 0,Y 137.816,Z 521.9,A -85,B 0,C 180,E1 -25724.372,E2 -25724.372} C_VEL
LIN {X 0,Y 137.22,Z 520.588,A -85,B 0,C 180,E1 -25725.537,E2 -25725.537} C_VEL
LIN {X 0,Y 134.899,Z 518.425,A -85,B 0,C 180,E1 -25730.621,E2 -25730.621} C_VEL
LIN {X 0,Y 133.642,Z 515.501,A -85,B 0,C 180,E1 -25736.604,E2 -25736.604} C_VEL
LIN {X 0,Y 133.45,Z 514.931,A -85,B 0,C 180,E1 -25739.995,E2 -25739.995} C_VEL
LIN {X 0,Y 133.782,Z 515.883,A -85,B 0,C 180,E1 -25744.892,E2 -25744.892} C_VEL
LIN {X 0,Y 136.419,Z 520.128,A -85,B 0,C 180,E1 -25753.4,E2 -25753.4} C_VEL
LIN {X 0,Y 137.347,Z 520.841,A -85,B 0,C 180,E1 -25755.103,E2 -25755.103} C_VEL
LIN {X 0,Y 139.436,Z 524.322,A -85,B 0,C 180,E1 -25758.609,E2 -25758.609} C_VEL
LIN {X 0,Y 141.05,Z 526.132,A -85,B 0,C 180,E1 -25760.745,E2 -25760.745} C_VEL
LIN {X 0,Y 143.808,Z 529.917,A -85,B 0,C 180,E1 -25763.964,E2 -25763.964} C_VEL
LIN {X 0,Y 147.622,Z 535.619,A -85,B 0,C 180,E1 -25767.722,E2 -25767.722} C_VEL
LIN {X 0,Y 151.794,Z 542.272,A -85,B 0,C 180,E1 -25771.21,E2 -25771.21} C_VEL
LIN {X 0,Y 156.813,Z 551.166,A -85,B 0,C 180,E1 -25774.844,E2 -25774.844} C_VEL
LIN {X 0,Y 161.014,Z 559.574,A -85,B 0,C 180,E1 -25777.562,E2 -25777.562} C_VEL
LIN {X 0,Y 165.113,Z 569.176,A -85,B 0,C 180,E1 -25780.029,E2 -25780.029} C_VEL
LIN {X 0,Y 172.438,Z 589.225,A -85,B 0,C 180,E1 -25784.156,E2 -25784.156} C_VEL
LIN {X 0,Y 176.198,Z 598.589,A -85,B 0,C 180,E1 -25786.293,E2 -25786.293} C_VEL
LIN {X 0,Y 180.11,Z 607.578,A -85,B 0,C 180,E1 -25788.598,E2 -25788.598} C_VEL
LIN {X 0,Y 184.855,Z 617.261,A -85,B 0,C 180,E1 -25791.385,E2 -25791.385} C_VEL
LIN {X 0,Y 190.231,Z 626.478,A -85,B 0,C 180,E1 -25794.362,E2 -25794.362} C_VEL
LIN {X 0,Y 196.476,Z 635.432,A -85,B 0,C 180,E1 -25797.551,E2 -25797.551} C_VEL
LIN {X 0,Y 204.51,Z 644.864,A -85,B 0,C 180,E1 -25801.242,E2 -25801.242} C_VEL
LIN {X 0,Y 212.902,Z 652.656,A -85,B 0,C 180,E1 -25804.588,E2 -25804.588} C_VEL
LIN {X 0,Y 223.357,Z 660.23,A -85,B 0,C 180,E1 -25808.148,E2 -25808.148} C_VEL
LIN {X 0,Y 236.499,Z 667.688,A -85,B 0,C 180,E1 -25811.967,E2 -25811.967} C_VEL
LIN {X 0,Y 249.199,Z 673.722,A -85,B 0,C 180,E1 -25815.296,E2 -25815.296} C_VEL
LIN {X 0,Y 258.813,Z 678.001,A -85,B 0,C 180,E1 -25817.827,E2 -25817.827} C_VEL
LIN {X 0,Y 267.092,Z 681.69,A -85,B 0,C 180,E1 -25820.198,E2 -25820.198} C_VEL
LIN {X 0,Y 270.246,Z 683.09,A -85,B 0,C 180,E1 -25821.179,E2 -25821.179} C_VEL
LIN {X 0,Y 274.127,Z 684.971,A -85,B 0,C 180,E1 -25822.635,E2 -25822.635} C_VEL
LIN {X 0,Y 277.361,Z 686.668,A -85,B 0,C 180,E1 -25824.183,E2 -25824.183} C_VEL
LIN {X 0,Y 281.61,Z 688.585,A -85,B 0,C 180,E1 -25826.569,E2 -25826.569} C_VEL
LIN {X 0,Y 282.416,Z 688.9,A -85,B 0,C 180,E1 -25827.147,E2 -25827.147} C_VEL
LIN {X 0,Y 283.856,Z 689.461,A -85,B 0,C 180,E1 -25828.581,E2 -25828.581} C_VEL
LIN {X 0,Y 284.632,Z 689.645,A -85,B 0,C 180,E1 -25830,E2 -25830} C_VEL
LIN {X 0,Y 283.862,Z 689.461,A -85,B 0,C 180,E1 -25831.419,E2 -25831.419} C_VEL
LIN {X 0,Y 282.407,Z 688.901,A -85,B 0,C 180,E1 -25832.853,E2 -25832.853} C_VEL
LIN {X 0,Y 280.053,Z 687.982,A -85,B 0,C 180,E1 -25834.318,E2 -25834.318} C_VEL
LIN {X 0,Y 275.882,Z 685.901,A -85,B 0,C 180,E1 -25836.556,E2 -25836.556} C_VEL
LIN {X 0,Y 274.088,Z 684.972,A -85,B 0,C 180,E1 -25837.366,E2 -25837.366} C_VEL
LIN {X 0,Y 269.606,Z 682.847,A -85,B 0,C 180,E1 -25838.998,E2 -25838.998} C_VEL
LIN {X 0,Y 261.365,Z 679.146,A -85,B 0,C 180,E1 -25841.478,E2 -25841.478} C_VEL
LIN {X 0,Y 253.155,Z 675.47,A -85,B 0,C 180,E1 -25843.687,E2 -25843.687} C_VEL
LIN {X 0,Y 240.334,Z 669.617,A -85,B 0,C 180,E1 -25847.003,E2 -25847.003} C_VEL
LIN {X 0,Y 225.92,Z 661.841,A -85,B 0,C 180,E1 -25851.063,E2 -25851.063} C_VEL
LIN {X 0,Y 214.415,Z 653.84,A -85,B 0,C 180,E1 -25854.871,E2 -25854.871} C_VEL
LIN {X 0,Y 206.668,Z 647.035,A -85,B 0,C 180,E1 -25857.859,E2 -25857.859} C_VEL
LIN {X 0,Y 199.669,Z 639.417,A -85,B 0,C 180,E1 -25860.936,E2 -25860.936} C_VEL
LIN {X 0,Y 192.541,Z 630.059,A -85,B 0,C 180,E1 -25864.406,E2 -25864.406} C_VEL
LIN {X 0,Y 186.463,Z 620.291,A -85,B 0,C 180,E1 -25867.679,E2 -25867.679} C_VEL
LIN {X 0,Y 181.99,Z 611.477,A -85,B 0,C 180,E1 -25870.305,E2 -25870.305} C_VEL
LIN {X 0,Y 177.438,Z 601.474,A -85,B 0,C 180,E1 -25872.992,E2 -25872.992} C_VEL
LIN {X 0,Y 173.059,Z 590.759,A -85,B 0,C 180,E1 -25875.536,E2 -25875.536} C_VEL
LIN {X 0,Y 167.494,Z 575.653,A -85,B 0,C 180,E1 -25878.589,E2 -25878.589} C_VEL
LIN {X 0,Y 163.656,Z 565.58,A -85,B 0,C 180,E1 -25880.831,E2 -25880.831} C_VEL
LIN {X 0,Y 158.972,Z 555.314,A -85,B 0,C 180,E1 -25883.732,E2 -25883.732} C_VEL
LIN {X 0,Y 153.947,Z 545.997,A -85,B 0,C 180,E1 -25887.165,E2 -25887.165} C_VEL
LIN {X 0,Y 150.091,Z 539.564,A -85,B 0,C 180,E1 -25890.145,E2 -25890.145} C_VEL
LIN {X 0,Y 146.466,Z 533.84,A -85,B 0,C 180,E1 -25893.35,E2 -25893.35} C_VEL
LIN {X 0,Y 143.491,Z 529.608,A -85,B 0,C 180,E1 -25896.363,E2 -25896.363} C_VEL
LIN {X 0,Y 140.441,Z 525.327,A -85,B 0,C 180,E1 -25900.047,E2 -25900.047} C_VEL
LIN {X 0,Y 137.954,Z 522.161,A -85,B 0,C 180,E1 -25903.733,E2 -25903.733} C_VEL
LIN {X 0,Y 137.212,Z 520.566,A -85,B 0,C 180,E1 -25905.166,E2 -25905.166} C_VEL
LIN {X 0,Y 134.941,Z 518.527,A -85,B 0,C 180,E1 -25910.095,E2 -25910.095} C_VEL
LIN {X 0,Y 133.636,Z 515.523,A -85,B 0,C 180,E1 -25916.235,E2 -25916.235} C_VEL
LIN {X 0,Y 133.45,Z 514.929,A -85,B 0,C 180,E1 -25920.005,E2 -25920.005} C_VEL
LIN {X 0,Y 133.783,Z 515.907,A -85,B 0,C 180,E1 -25924.524,E2 -25924.524} C_VEL
LIN {X 0,Y 136.431,Z 520.106,A -85,B 0,C 180,E1 -25933.029,E2 -25933.029} C_VEL
LIN {X 0,Y 137.357,Z 520.854,A -85,B 0,C 180,E1 -25934.732,E2 -25934.732} C_VEL
LIN {X 0,Y 139.409,Z 524.277,A -85,B 0,C 180,E1 -25938.18,E2 -25938.18} C_VEL
LIN {X 0,Y 140.964,Z 525.971,A -85,B 0,C 180,E1 -25940.24,E2 -25940.24} C_VEL
LIN {X 0,Y 144.587,Z 531.119,A -85,B 0,C 180,E1 -25944.408,E2 -25944.408} C_VEL
LIN {X 0,Y 147.742,Z 535.832,A -85,B 0,C 180,E1 -25947.445,E2 -25947.445} C_VEL
LIN {X 0,Y 150.451,Z 540.163,A -85,B 0,C 180,E1 -25949.762,E2 -25949.762} C_VEL
LIN {X 0,Y 153.997,Z 547.786,A -85,B 0,C 180,E1 -25952.626,E2 -25952.626} C_VEL
LIN {X 0,Y 158.797,Z 559.78,A -85,B 0,C 180,E1 -25956.128,E2 -25956.128} C_VEL
LIN {X 0,Y 161.018,Z 566.501,A -85,B 0,C 180,E1 -25957.671,E2 -25957.671} C_VEL
LIN {X 0,Y 158.548,Z 596.386,A -85,B 0,C 180,E1 -25958.804,E2 -25958.804} C_VEL
LIN {X 0,Y 156.882,Z 607.423,A -85,B 0,C 180,E1 -25959.478,E2 -25959.478} C_VEL
LIN {X 0,Y 154.474,Z 618.066,A -85,B 0,C 180,E1 -25960.354,E2 -25960.354} C_VEL
LIN {X 0,Y 150.862,Z 630.512,A -85,B 0,C 180,E1 -25961.81,E2 -25961.81} C_VEL
LIN {X 0,Y 146.728,Z 641.46,A -85,B 0,C 180,E1 -25963.577,E2 -25963.577} C_VEL
LIN {X 0,Y 142.25,Z 651.494,A -85,B 0,C 180,E1 -25965.745,E2 -25965.745} C_VEL
LIN {X 0,Y 138.466,Z 658.909,A -85,B 0,C 180,E1 -25967.739,E2 -25967.739} C_VEL
LIN {X 0,Y 133.491,Z 667.701,A -85,B 0,C 180,E1 -25970.819,E2 -25970.819} C_VEL
LIN {X 0,Y 129.827,Z 673.689,A -85,B 0,C 180,E1 -25973.454,E2 -25973.454} C_VEL
LIN {X 0,Y 125.835,Z 679.893,A -85,B 0,C 180,E1 -25976.912,E2 -25976.912} C_VEL
LIN {X 0,Y 122.153,Z 685.277,A -85,B 0,C 180,E1 -25980.723,E2 -25980.723} C_VEL
LIN {X 0,Y 118.412,Z 690.371,A -85,B 0,C 180,E1 -25985.452,E2 -25985.452} C_VEL
LIN {X 0,Y 115.502,Z 694.338,A -85,B 0,C 180,E1 -25990.448,E2 -25990.448} C_VEL
LIN {X 0,Y 113.62,Z 697.282,A -85,B 0,C 180,E1 -25995.675,E2 -25995.675} C_VEL
LIN {X 0,Y 112.759,Z 698.789,A -85,B 0,C 180,E1 -25999.223,E2 -25999.223} C_VEL
LIN {X 0,Y 112.135,Z 700.328,A -85,B 0,C 180,E1 -26006.407,E2 -26006.407} C_VEL
LIN {X 0,Y 112.257,Z 700.614,A -85,B 0,C 180,E1 -26010,E2 -26010} C_VEL
LIN {X 0,Y 112.272,Z 699.724,A -85,B 0,C 180,E1 -26017.192,E2 -26017.192} C_VEL
LIN {X 0,Y 112.762,Z 698.789,A -85,B 0,C 180,E1 -26020.776,E2 -26020.776} C_VEL
LIN {X 0,Y 114.778,Z 695.43,A -85,B 0,C 180,E1 -26027.827,E2 -26027.827} C_VEL
LIN {X 0,Y 117.35,Z 691.799,A -85,B 0,C 180,E1 -26032.909,E2 -26032.909} C_VEL
LIN {X 0,Y 120.766,Z 687.065,A -85,B 0,C 180,E1 -26037.746,E2 -26037.746} C_VEL
LIN {X 0,Y 124.977,Z 681.112,A -85,B 0,C 180,E1 -26042.275,E2 -26042.275} C_VEL
LIN {X 0,Y 128.162,Z 676.313,A -85,B 0,C 180,E1 -26045.154,E2 -26045.154} C_VEL
LIN {X 0,Y 131.629,Z 670.821,A -85,B 0,C 180,E1 -26047.88,E2 -26047.88} C_VEL
LIN {X 0,Y 136.435,Z 662.608,A -85,B 0,C 180,E1 -26051.054,E2 -26051.054} C_VEL
LIN {X 0,Y 140.611,Z 654.787,A -85,B 0,C 180,E1 -26053.412,E2 -26053.412} C_VEL
LIN {X 0,Y 144.456,Z 646.708,A -85,B 0,C 180,E1 -26055.359,E2 -26055.359} C_VEL
LIN {X 0,Y 148.459,Z 636.953,A -85,B 0,C 180,E1 -26057.202,E2 -26057.202} C_VEL
LIN {X 0,Y 151.396,Z 628.566,A -85,B 0,C 180,E1 -26058.464,E2 -26058.464} C_VEL
LIN {X 0,Y 154.424,Z 618.064,A -85,B 0,C 180,E1 -26059.668,E2 -26059.668} C_VEL
LIN {X 0,Y 156.684,Z 608.291,A -85,B 0,C 180,E1 -26060.482,E2 -26060.482} C_VEL
LIN {X 0,Y 158.449,Z 597.44,A -85,B 0,C 180,E1 -26061.127,E2 -26061.127} C_VEL
LIN {X 0,Y 160.448,Z 574.242,A -85,B 0,C 180,E1 -26062.039,E2 -26062.039} C_VEL
LIN {X 0,Y 161.024,Z 566.44,A -85,B 0,C 180,E1 -26062.331,E2 -26062.331} C_VEL
LIN {X 0,Y 157.523,Z 556.435,A -85,B 0,C 180,E1 -26064.764,E2 -26064.764} C_VEL
LIN {X 0,Y 152.945,Z 545.45,A -85,B 0,C 180,E1 -26068.193,E2 -26068.193} C_VEL
LIN {X 0,Y 150.929,Z 541.166,A -85,B 0,C 180,E1 -26069.832,E2 -26069.832} C_VEL
LIN {X 0,Y 149.751,Z 539.443,A -85,B 0,C 180,E1 -26070.774,E2 -26070.774} C_VEL
LIN {X 0,Y 147.686,Z 538.439,A -85,B 0,C 180,E1 -26072.33,E2 -26072.33} C_VEL
LIN {X 0,Y 143.499,Z 537.852,A -85,B 0,C 180,E1 -26075.749,E2 -26075.749} C_VEL
LIN {X 0,Y 142.084,Z 536.551,A -85,B 0,C 180,E1 -26077.2,E2 -26077.2} C_VEL
LIN {X 0,Y 138.675,Z 531.77,A -85,B 0,C 180,E1 -26081.529,E2 -26081.529} C_VEL
LIN {X 0,Y 136.211,Z 528.148,A -85,B 0,C 180,E1 -26085.618,E2 -26085.618} C_VEL
LIN {X 0,Y 135.768,Z 527.366,A -85,B 0,C 180,E1 -26086.525,E2 -26086.525} C_VEL
LIN {X 0,Y 133.294,Z 524.313,A -85,B 0,C 180,E1 -26093.182,E2 -26093.182} C_VEL
LIN {X 0,Y 132.732,Z 522.494,A -85,B 0,C 180,E1 -26096.96,E2 -26096.96} C_VEL
LIN {X 0,Y 132.583,Z 521.991,A -85,B 0,C 180,E1 -26099.995,E2 -26099.995} C_VEL
LIN {X 0,Y 132.832,Z 522.81,A -85,B 0,C 180,E1 -26104.357,E2 -26104.357} C_VEL
LIN {X 0,Y 135.206,Z 526.992,A -85,B 0,C 180,E1 -26112.758,E2 -26112.758} C_VEL
LIN {X 0,Y 136.032,Z 527.739,A -85,B 0,C 180,E1 -26114.392,E2 -26114.392} C_VEL
LIN {X 0,Y 138.296,Z 531.416,A -85,B 0,C 180,E1 -26118.33,E2 -26118.33} C_VEL
LIN {X 0,Y 139.39,Z 532.721,A -85,B 0,C 180,E1 -26119.854,E2 -26119.854} C_VEL
LIN {X 0,Y 142.528,Z 537.389,A -85,B 0,C 180,E1 -26123.71,E2 -26123.71} C_VEL
LIN {X 0,Y 145.471,Z 541.982,A -85,B 0,C 180,E1 -26126.747,E2 -26126.747} C_VEL
LIN {X 0,Y 149.381,Z 548.552,A -85,B 0,C 180,E1 -26130.23,E2 -26130.23} C_VEL
LIN {X 0,Y 153.689,Z 556.517,A -85,B 0,C 180,E1 -26133.57,E2 -26133.57} C_VEL
LIN {X 0,Y 157.827,Z 565.255,A -85,B 0,C 180,E1 -26136.45,E2 -26136.45} C_VEL
LIN {X 0,Y 161.769,Z 575.186,A -85,B 0,C 180,E1 -26139.007,E2 -26139.007} C_VEL
LIN {X 0,Y 167.468,Z 591.85,A -85,B 0,C 180,E1 -26142.581,E2 -26142.581} C_VEL
